C05412=1045.140,185.650,-96.102,170.888,38.031,157.175
C05413=1045.134,185.400,-96.077,170.885,38.029,157.175
C05414=1045.128,185.152,-96.053,170.883,38.027,157.174
C05415=1045.123,184.903,-96.029,170.881,38.025,157.174
C05416=1045.116,184.654,-96.006,170.877,38.023,157.173
C05417=1045.110,184.406,-95.982,170.875,38.021,157.173
C05418=1045.105,184.156,-95.958,170.873,38.019,157.173
C05419=1045.098,183.908,-95.934,170.870,38.018,157.172
C05420=1045.093,183.659,-95.909,170.868,38.017,157.172
C05421=1045.087,183.410,-95.886,170.865,38.015,157.172
C05422=1045.079,183.161,-95.863,170.863,38.013,157.171
C05423=1045.073,182.913,-95.839,170.860,38.011,157.171
C05424=1045.067,182.664,-95.815,170.858,38.010,157.171
C05425=1045.061,182.415,-95.792,170.856,38.008,157.170
C05426=1045.054,182.166,-95.768,170.852,38.007,157.170
C05427=1045.048,181.918,-95.745,170.850,38.005,157.169
C05428=1045.042,181.668,-95.721,170.848,38.004,157.169
C05429=1045.036,181.420,-95.698,170.846,38.002,157.169
C05430=1045.029,181.171,-95.674,170.843,38.000,157.168
C05431=1045.024,180.922,-95.651,170.840,37.999,157.168
C05432=1045.018,180.674,-95.627,170.838,37.997,157.168
C05433=1045.011,180.424,-95.604,170.835,37.996,157.167
C05434=1045.005,180.176,-95.580,170.833,37.994,157.167
C05435=1044.999,179.927,-95.556,170.831,37.993,157.167
C05436=1044.993,179.678,-95.533,170.828,37.991,157.166
C05437=1044.986,179.429,-95.510,170.825,37.989,157.166
C05438=1044.980,179.180,-95.487,170.823,37.988,157.165
C05439=1044.974,178.932,-95.463,170.821,37.986,157.165
C05440=1044.967,178.682,-95.440,170.818,37.984,157.165
C05441=1044.961,178.434,-95.416,170.815,37.983,157.164
C05442=1044.955,178.185,-95.393,170.813,37.982,157.164
C05443=1044.949,177.936,-95.369,170.811,37.980,157.164
C05444=1044.943,177.687,-95.346,170.808,37.979,157.163
C05445=1044.937,177.438,-95.322,170.806,37.977,157.163
C05446=1044.931,177.190,-95.299,170.804,37.975,157.163
C05447=1044.925,176.941,-95.276,170.802,37.974,157.162
C05448=1044.918,176.692,-95.253,170.798,37.972,157.162
C05449=1044.912,176.444,-95.229,170.796,37.970,157.161
C05450=1044.905,176.194,-95.206,170.794,37.969,157.161
C05451=1044.899,175.946,-95.182,170.791,37.967,157.161
C05452=1044.894,175.697,-95.159,170.789,37.966,157.160
C05453=1044.887,175.447,-95.136,170.787,37.965,157.160
C05454=1044.881,175.199,-95.112,170.784,37.963,157.160
C05455=1044.876,174.950,-95.089,170.781,37.961,157.159
C05456=1044.869,174.702,-95.066,170.779,37.960,157.159
C05457=1044.862,174.453,-95.043,170.777,37.958,157.159
C05458=1044.857,174.204,-95.020,170.774,37.956,157.158
C05459=1044.850,173.919,-94.993,170.772,37.955,157.158
C05460=1044.843,173.634,-94.967,170.769,37.953,157.158
C05461=1044.836,173.349,-94.940,170.766,37.951,157.157
C05462=1044.829,173.064,-94.913,170.763,37.949,157.157
C05463=1044.823,172.815,-94.891,170.761,37.947,157.156
C05464=1044.817,172.567,-94.868,170.759,37.946,157.156
C05465=1044.810,172.318,-94.844,170.756,37.945,157.156
C05466=1044.804,172.069,-94.821,170.754,37.943,157.155
C05467=1044.799,171.820,-94.798,170.752,37.942,157.155
C05468=1044.793,171.572,-94.774,170.749,37.940,157.155
C05469=1044.787,171.323,-94.751,170.747,37.938,157.154
C05470=1044.780,171.073,-94.728,170.744,37.937,157.154
C05471=1044.774,170.824,-94.705,170.742,37.935,157.154
C05472=1044.768,170.576,-94.682,170.739,37.933,157.153
C05473=1044.762,170.327,-94.659,170.737,37.932,157.153
C05474=1044.757,170.078,-94.636,170.735,37.930,157.153
C05475=1044.750,169.829,-94.613,170.733,37.929,157.152
C05476=1044.744,169.580,-94.590,170.730,37.927,157.152
C05477=1044.738,169.331,-94.567,170.728,37.926,157.151
C05478=1044.732,169.083,-94.544,170.726,37.925,157.151
C05479=1044.726,168.834,-94.521,170.723,37.923,157.151
C05480=1044.720,168.585,-94.497,170.721,37.921,157.150
C05481=1044.714,168.336,-94.474,170.719,37.920,157.150
C05482=1044.708,168.087,-94.452,170.717,37.918,157.150
C05483=1044.702,167.838,-94.429,170.714,37.916,157.149
C05484=1044.696,167.589,-94.406,170.712,37.915,157.149
C05485=1044.690,167.341,-94.383,170.709,37.913,157.149
C05486=1044.685,167.092,-94.360,170.707,37.912,157.148
C05487=1044.679,166.843,-94.337,170.704,37.910,157.148
C05488=1044.672,166.594,-94.314,170.702,37.909,157.148
C05489=1044.666,166.345,-94.291,170.700,37.907,157.147
C05490=1044.660,166.096,-94.268,170.697,37.906,157.147
C05491=1044.655,165.847,-94.245,170.695,37.904,157.147
C05492=1044.649,165.598,-94.222,170.693,37.903,157.146
C05493=1044.642,165.350,-94.200,170.691,37.901,157.146
C05494=1044.637,165.101,-94.177,170.688,37.900,157.146
C05495=1044.631,164.852,-94.154,170.686,37.898,157.145
C05496=1044.625,164.603,-94.131,170.684,37.896,157.145
C05497=1044.619,164.354,-94.108,170.682,37.895,157.145
C05498=1044.613,164.106,-94.086,170.679,37.893,157.144
C05499=1044.607,163.857,-94.063,170.677,37.891,157.144
C05500=1044.601,163.607,-94.039,170.675,37.890,157.144
C05501=1044.595,163.358,-94.016,170.672,37.889,157.143
C05502=1044.589,163.109,-93.993,170.670,37.887,157.143
C05503=1044.583,162.861,-93.971,170.668,37.886,157.143
C05504=1044.577,162.612,-93.948,170.666,37.884,157.142
C05505=1044.572,162.363,-93.925,170.663,37.883,157.142
C05506=1044.566,162.114,-93.902,170.661,37.881,157.142
C05507=1044.560,161.865,-93.881,170.659,37.879,157.141
C05508=1044.554,161.616,-93.858,170.657,37.878,157.141
C05509=1044.548,161.367,-93.835,170.654,37.876,157.140
C05510=1044.542,161.118,-93.812,170.652,37.875,157.140
C05511=1044.537,160.869,-93.789,170.650,37.873,157.140
C05512=1044.530,160.621,-93.767,170.647,37.871,157.139
C05513=1044.525,160.372,-93.744,170.645,37.870,157.139
C05514=1044.519,160.122,-93.721,170.643,37.868,157.139
C05515=1044.513,159.874,-93.699,170.641,37.867,157.138
C05516=1044.506,159.625,-93.677,170.638,37.865,157.138
C05517=1044.501,159.376,-93.654,170.636,37.864,157.138
C05518=1044.494,159.127,-93.632,170.634,37.863,157.138
C05519=1044.489,158.878,-93.609,170.632,37.861,157.137
C05520=1044.482,158.629,-93.587,170.629,37.860,157.137
C05521=1044.476,158.380,-93.565,170.627,37.858,157.137
C05522=1044.470,158.131,-93.542,170.625,37.857,157.136
C05523=1044.463,157.846,-93.517,170.623,37.855,157.136
C05524=1044.456,157.561,-93.491,170.620,37.854,157.136
C05525=1044.449,157.275,-93.466,170.617,37.852,157.135
C05526=1044.441,156.990,-93.440,170.615,37.851,157.135
C05527=1044.436,156.741,-93.418,170.613,37.850,157.135
C05528=1044.430,156.492,-93.395,170.610,37.848,157.134
C05529=1044.423,156.243,-93.374,170.608,37.847,157.134
C05530=1044.418,155.994,-93.351,170.606,37.845,157.134
C05531=1044.411,155.745,-93.328,170.604,37.844,157.133
C05532=1044.405,155.496,-93.307,170.601,37.842,157.133
C05533=1044.400,155.248,-93.284,170.599,37.841,157.133
C05534=1044.394,154.999,-93.262,170.597,37.839,157.132
C05535=1044.388,154.750,-93.239,170.595,37.838,157.132
C05536=1044.382,154.501,-93.218,170.592,37.837,157.132
C05537=1044.375,154.252,-93.196,170.590,37.835,157.131
C05538=1044.369,154.003,-93.174,170.588,37.834,157.131
C05539=1044.363,153.754,-93.151,170.586,37.832,157.131
C05540=1044.357,153.505,-93.129,170.583,37.831,157.131
C05541=1044.351,153.256,-93.107,170.581,37.829,157.130
C05542=1044.345,153.007,-93.085,170.579,37.828,157.130
C05543=1044.338,152.758,-93.063,170.577,37.827,157.130
C05544=1044.333,152.509,-93.041,170.574,37.825,157.129
C05545=1044.326,152.260,-93.018,170.572,37.824,157.129
C05546=1044.320,152.011,-92.997,170.570,37.823,157.129
C05547=1044.314,151.762,-92.974,170.569,37.821,157.128
C05548=1044.308,151.513,-92.952,170.567,37.820,157.128
C05549=1044.302,151.264,-92.931,170.564,37.819,157.128
C05550=1044.296,151.016,-92.909,170.562,37.817,157.127
C05551=1044.290,150.767,-92.887,170.560,37.816,157.127
C05552=1044.284,150.518,-92.865,170.558,37.815,157.127
C05553=1044.278,150.269,-92.842,170.555,37.813,157.126
C05554=1044.272,150.019,-92.821,170.553,37.812,157.126
C05555=1044.266,149.771,-92.798,170.551,37.810,157.126
C05556=1044.259,149.522,-92.777,170.549,37.809,157.126
C05557=1044.253,149.272,-92.755,170.546,37.808,157.125
C05558=1044.247,149.024,-92.733,170.544,37.806,157.125
C05559=1044.242,148.775,-92.711,170.542,37.805,157.125
C05560=1044.236,148.526,-92.689,170.540,37.803,157.124
C05561=1044.230,148.277,-92.668,170.538,37.802,157.124
C05562=1044.223,148.028,-92.645,170.535,37.801,157.124
C05563=1044.217,147.779,-92.624,170.533,37.799,157.123
C05564=1044.211,147.530,-92.602,170.532,37.798,157.123
C05565=1044.205,147.280,-92.580,170.530,37.797,157.123
C05566=1044.199,147.032,-92.558,170.527,37.796,157.123
C05567=1044.193,146.783,-92.537,170.525,37.794,157.122
C05568=1044.186,146.534,-92.515,170.523,37.793,157.122
C05569=1044.180,146.285,-92.493,170.521,37.792,157.122
C05570=1044.174,146.036,-92.472,170.518,37.790,157.122
C05571=1044.168,145.787,-92.449,170.516,37.789,157.121
C05572=1044.161,145.538,-92.428,170.514,37.787,157.121
C05573=1044.156,145.289,-92.407,170.512,37.786,157.121
C05574=1044.150,145.040,-92.385,170.510,37.785,157.120
C05575=1044.144,144.791,-92.363,170.507,37.784,157.120
C05576=1044.137,144.542,-92.342,170.505,37.783,157.120
C05577=1044.131,144.293,-92.320,170.503,37.781,157.119
C05578=1044.125,144.045,-92.298,170.502,37.780,157.119
C05579=1044.119,143.795,-92.276,170.499,37.778,157.119
C05580=1044.113,143.546,-92.255,170.497,37.777,157.119
C05581=1044.107,143.297,-92.233,170.495,37.775,157.118
C05582=1044.101,143.048,-92.211,170.493,37.774,157.118
C05583=1044.095,142.799,-92.190,170.491,37.773,157.118
C05584=1044.089,142.550,-92.169,170.488,37.772,157.117
C05585=1044.082,142.301,-92.148,170.486,37.771,157.117
C05586=1044.076,142.052,-92.126,170.484,37.769,157.117
C05587=1044.069,141.767,-92.101,170.482,37.768,157.117
C05588=1044.063,141.481,-92.076,170.479,37.766,157.116
C05589=1044.056,141.195,-92.051,170.477,37.765,157.116
C05590=1044.048,140.909,-92.027,170.475,37.763,157.116
C05591=1044.043,140.661,-92.006,170.473,37.762,157.115
C05592=1044.037,140.412,-91.984,170.470,37.761,157.115
C05593=1044.030,140.162,-91.963,170.468,37.759,157.115
C05594=1044.024,139.913,-91.941,170.466,37.758,157.114
C05595=1044.019,139.665,-91.920,170.464,37.757,157.114
C05596=1044.013,139.416,-91.898,170.462,37.755,157.114
C05597=1044.006,139.166,-91.877,170.459,37.754,157.114
C05598=1043.999,138.917,-91.856,170.458,37.753,157.113
C05599=1043.994,138.669,-91.834,170.456,37.751,157.113
C05600=1043.988,138.420,-91.813,170.454,37.750,157.113
C05601=1043.982,138.170,-91.791,170.451,37.749,157.112
C05602=1043.975,137.922,-91.770,170.449,37.748,157.112
C05603=1043.969,137.672,-91.749,170.447,37.746,157.112
C05604=1043.963,137.423,-91.728,170.445,37.745,157.112
C05605=1043.957,137.174,-91.706,170.443,37.744,157.111
C05606=1043.951,136.926,-91.685,170.441,37.742,157.111
C05607=1043.945,136.677,-91.664,170.439,37.741,157.111
C05608=1043.939,136.427,-91.643,170.437,37.740,157.110
C05609=1043.933,136.179,-91.622,170.435,37.739,157.110
C05610=1043.926,135.929,-91.601,170.433,37.737,157.110
C05611=1043.920,135.680,-91.579,170.430,37.736,157.110
C05612=1043.914,135.431,-91.557,170.428,37.735,157.109
C05613=1043.908,135.182,-91.537,170.426,37.734,157.109
C05614=1043.902,134.933,-91.516,170.425,37.733,157.109
C05615=1043.896,134.684,-91.494,170.422,37.731,157.109
C05616=1043.889,134.436,-91.473,170.420,37.730,157.108
C05617=1043.884,134.186,-91.453,170.418,37.729,157.108
C05618=1043.878,133.937,-91.431,170.416,37.727,157.108
C05619=1043.871,133.688,-91.410,170.414,37.726,157.107
C05620=1043.865,133.439,-91.389,170.411,37.725,157.107
C05621=1043.860,133.190,-91.368,170.410,37.724,157.107
C05622=1043.853,132.941,-91.347,170.408,37.723,157.107
C05623=1043.847,132.692,-91.325,170.406,37.721,157.106
C05624=1043.841,132.443,-91.305,170.404,37.720,157.106
C05625=1043.834,132.194,-91.284,170.401,37.718,157.106
C05626=1043.828,131.945,-91.262,170.399,37.717,157.106
C05627=1043.823,131.696,-91.242,170.397,37.716,157.105
C05628=1043.816,131.447,-91.221,170.396,37.715,157.105
C05629=1043.811,131.198,-91.200,170.394,37.714,157.105
C05630=1043.804,130.949,-91.179,170.391,37.712,157.104
C05631=1043.798,130.699,-91.157,170.389,37.711,157.104
C05632=1043.792,130.451,-91.137,170.387,37.710,157.104
C05633=1043.785,130.202,-91.116,170.385,37.709,157.104
C05634=1043.779,129.952,-91.095,170.383,37.708,157.103
C05635=1043.773,129.704,-91.075,170.381,37.707,157.103
C05636=1043.767,129.454,-91.054,170.379,37.705,157.103
C05637=1043.760,129.205,-91.033,170.377,37.704,157.103
C05638=1043.754,128.956,-91.013,170.375,37.703,157.102
C05639=1043.748,128.707,-90.991,170.373,37.702,157.102
C05640=1043.742,128.458,-90.971,170.370,37.701,157.102
C05641=1043.735,128.209,-90.950,170.368,37.699,157.102
C05642=1043.729,127.959,-90.929,170.367,37.698,157.101
C05643=1043.723,127.711,-90.909,170.365,37.697,157.101
C05644=1043.716,127.462,-90.888,170.363,37.696,157.101
C05645=1043.711,127.213,-90.868,170.360,37.695,157.101
C05646=1043.704,126.964,-90.847,170.358,37.693,157.100
C05647=1043.698,126.714,-90.826,170.356,37.692,157.100
C05648=1043.692,126.466,-90.805,170.354,37.691,157.100
C05649=1043.685,126.216,-90.785,170.353,37.690,157.100
C05650=1043.680,125.967,-90.764,170.350,37.689,157.099
C05651=1043.672,125.681,-90.740,170.348,37.687,157.099
C05652=1043.665,125.396,-90.716,170.346,37.686,157.099
C05653=1043.658,125.110,-90.692,170.343,37.685,157.098
C05654=1043.651,124.824,-90.669,170.341,37.683,157.098
C05655=1043.645,124.575,-90.649,170.339,37.682,157.098
C05656=1043.639,124.325,-90.628,170.337,37.681,157.098
C05657=1043.633,124.077,-90.607,170.335,37.680,157.097
C05658=1043.626,123.828,-90.587,170.333,37.679,157.097
C05659=1043.620,123.578,-90.566,170.331,37.677,157.097
C05660=1043.614,123.330,-90.545,170.328,37.676,157.097
C05661=1043.607,123.080,-90.525,170.327,37.675,157.096
C05662=1043.602,122.831,-90.504,170.325,37.674,157.096
C05663=1043.595,122.582,-90.484,170.323,37.673,157.096
C05664=1043.589,122.333,-90.463,170.321,37.671,157.096
C05665=1043.583,122.085,-90.443,170.318,37.670,157.095
C05666=1043.577,121.835,-90.423,170.317,37.669,157.095
C05667=1043.571,121.587,-90.402,170.315,37.668,157.095
C05668=1043.564,121.337,-90.382,170.313,37.667,157.095
C05669=1043.559,121.088,-90.361,170.311,37.665,157.094
C05670=1043.553,120.838,-90.341,170.308,37.664,157.094
C05671=1043.547,120.590,-90.321,170.307,37.663,157.094
C05672=1043.540,120.340,-90.299,170.305,37.662,157.093
C05673=1043.534,120.092,-90.279,170.303,37.661,157.093
C05674=1043.528,119.842,-90.259,170.301,37.659,157.093
C05675=1043.523,119.593,-90.238,170.298,37.658,157.093
C05676=1043.516,119.345,-90.218,170.297,37.657,157.092
C05677=1043.510,119.095,-90.197,170.295,37.656,157.092
C05678=1043.504,118.846,-90.177,170.293,37.655,157.092
C05679=1043.498,118.597,-90.156,170.291,37.653,157.092
C05680=1043.492,118.348,-90.136,170.288,37.652,157.091
C05681=1043.485,118.098,-90.116,170.287,37.651,157.091
C05682=1043.480,117.849,-90.096,170.285,37.650,157.091
C05683=1043.474,117.601,-90.075,170.283,37.649,157.091
C05684=1043.467,117.351,-90.055,170.281,37.647,157.090
C05685=1043.461,117.103,-90.035,170.280,37.646,157.090
C05686=1043.456,116.854,-90.014,170.277,37.645,157.090
C05687=1043.449,116.604,-89.994,170.275,37.644,157.090
C05688=1043.443,116.355,-89.974,170.273,37.643,157.089
C05689=1043.437,116.105,-89.953,170.271,37.641,157.089
C05690=1043.431,115.857,-89.933,170.269,37.640,157.089
C05691=1043.425,115.608,-89.913,170.267,37.638,157.088
C05692=1043.419,115.358,-89.893,170.265,37.637,157.088
C05693=1043.413,115.110,-89.871,170.263,37.636,157.088
C05694=1043.407,114.861,-89.851,170.262,37.635,157.088
C05695=1043.401,114.611,-89.831,170.259,37.634,157.087
C05696=1043.395,114.363,-89.811,170.257,37.632,157.087
C05697=1043.389,114.113,-89.791,170.255,37.631,157.087
C05698=1043.383,113.864,-89.770,170.254,37.630,157.087
C05699=1043.377,113.615,-89.750,170.252,37.629,157.086
C05700=1043.371,113.366,-89.730,170.250,37.628,157.086
C05701=1043.364,113.117,-89.710,170.247,37.626,157.086
C05702=1043.358,112.868,-89.690,170.246,37.625,157.086
C05703=1043.353,112.619,-89.671,170.244,37.624,157.085
C05704=1043.346,112.369,-89.650,170.242,37.623,157.085
C05705=1043.340,112.120,-89.630,170.240,37.622,157.085
C05706=1043.333,111.871,-89.610,170.237,37.621,157.085
C05707=1043.327,111.622,-89.590,170.236,37.620,157.085
C05708=1043.321,111.373,-89.570,170.234,37.619,157.084
C05709=1043.315,111.124,-89.550,170.232,37.617,157.084
C05710=1043.309,110.875,-89.530,170.230,37.616,157.084
C05711=1043.303,110.626,-89.510,170.228,37.615,157.083
C05712=1043.296,110.376,-89.490,170.226,37.614,157.083
C05713=1043.290,110.127,-89.470,170.224,37.613,157.083
C05714=1043.284,109.878,-89.450,170.222,37.611,157.083
C05715=1043.278,109.592,-89.428,170.220,37.610,157.082
C05716=1043.270,109.306,-89.405,170.218,37.609,157.082
C05717=1043.263,109.020,-89.382,170.215,37.608,157.082
C05718=1043.256,108.734,-89.360,170.213,37.607,157.082
C05719=1043.250,108.485,-89.340,170.211,37.605,157.081
C05720=1043.243,108.236,-89.319,170.209,37.604,157.081
C05721=1043.237,107.986,-89.300,170.208,37.603,157.081
C05722=1043.231,107.737,-89.280,170.205,37.602,157.081
C05723=1043.224,107.488,-89.260,170.203,37.601,157.081
C05724=1043.218,107.239,-89.240,170.201,37.600,157.080
C05725=1043.212,106.990,-89.221,170.200,37.599,157.080
C05726=1043.206,106.741,-89.201,170.198,37.598,157.080
C05727=1043.200,106.492,-89.181,170.195,37.596,157.079
C05728=1043.194,106.243,-89.161,170.193,37.595,157.079
C05729=1043.188,105.993,-89.142,170.192,37.594,157.079
C05730=1043.181,105.745,-89.122,170.190,37.593,157.079
C05731=1043.175,105.495,-89.102,170.188,37.592,157.079
C05732=1043.169,105.246,-89.083,170.186,37.591,157.078
C05733=1043.163,104.997,-89.063,170.183,37.590,157.078
C05734=1043.157,104.748,-89.043,170.182,37.589,157.078
C05735=1043.151,104.498,-89.023,170.180,37.587,157.078
C05736=1043.144,104.250,-89.004,170.178,37.586,157.077
C05737=1043.138,104.000,-88.985,170.176,37.585,157.077
C05738=1043.132,103.751,-88.965,170.174,37.584,157.077
C05739=1043.126,103.502,-88.944,170.172,37.583,157.077
C05740=1043.120,103.253,-88.925,170.170,37.582,157.076
C05741=1043.113,103.004,-88.906,170.168,37.581,157.076
C05742=1043.108,102.755,-88.886,170.167,37.580,157.076
C05743=1043.102,102.506,-88.866,170.165,37.578,157.076
C05744=1043.095,102.256,-88.846,170.162,37.577,157.075
C05745=1043.089,102.007,-88.827,170.160,37.576,157.075
C05746=1043.083,101.758,-88.808,170.159,37.575,157.075
C05747=1043.077,101.509,-88.788,170.157,37.574,157.075
C05748=1043.071,101.260,-88.768,170.155,37.572,157.074
C05749=1043.065,101.010,-88.749,170.154,37.572,157.074
C05750=1043.059,100.761,-88.729,170.151,37.571,157.074
C05751=1043.052,100.512,-88.710,170.149,37.569,157.074
C05752=1043.046,100.263,-88.690,170.147,37.568,157.073
C05753=1043.041,100.014,-88.671,170.146,37.567,157.073
C05754=1043.033,99.765,-88.651,170.144,37.566,157.073
C05755=1043.028,99.515,-88.632,170.142,37.565,157.073
C05756=1043.021,99.267,-88.613,170.139,37.564,157.073
C05757=1043.015,99.017,-88.593,170.137,37.563,157.072
C05758=1043.008,98.769,-88.574,170.136,37.562,157.072
C05759=1043.002,98.519,-88.554,170.134,37.561,157.072
C05760=1042.996,98.269,-88.535,170.132,37.560,157.072
C05761=1042.990,98.021,-88.516,170.129,37.559,157.071
C05762=1042.984,97.771,-88.496,170.128,37.557,157.071
C05763=1042.977,97.523,-88.477,170.126,37.556,157.071
C05764=1042.972,97.273,-88.458,170.124,37.556,157.071
C05765=1042.965,97.023,-88.439,170.122,37.554,157.071
C05766=1042.959,96.775,-88.419,170.121,37.553,157.070
C05767=1042.952,96.525,-88.400,170.118,37.552,157.070
C05768=1042.946,96.276,-88.381,170.116,37.551,157.070
C05769=1042.940,96.028,-88.362,170.114,37.550,157.070
C05770=1042.934,95.778,-88.342,170.113,37.549,157.069
C05771=1042.928,95.529,-88.323,170.111,37.548,157.069
C05772=1042.921,95.279,-88.303,170.109,37.547,157.069
C05773=1042.915,95.030,-88.284,170.106,37.545,157.069
C05774=1042.909,94.781,-88.266,170.105,37.545,157.069
C05775=1042.903,94.532,-88.246,170.103,37.544,157.068
C05776=1042.896,94.283,-88.227,170.101,37.542,157.068
C05777=1042.891,94.034,-88.208,170.099,37.541,157.068
C05778=1042.884,93.784,-88.189,170.098,37.540,157.067
C05779=1042.877,93.499,-88.167,170.095,37.539,157.067
C05780=1042.871,93.212,-88.144,170.093,37.537,157.067
C05781=1042.863,92.926,-88.122,170.091,37.536,157.067
C05782=1042.856,92.640,-88.101,170.089,37.535,157.066
C05783=1042.850,92.391,-88.082,170.087,37.534,157.066
C05784=1042.844,92.142,-88.062,170.084,37.533,157.066
C05785=1042.837,91.893,-88.043,170.083,37.532,157.066
C05786=1042.831,91.644,-88.024,170.081,37.531,157.066
C05787=1042.825,91.394,-88.005,170.079,37.530,157.065
C05788=1042.819,91.145,-87.986,170.077,37.528,157.065
C05789=1042.813,90.897,-87.967,170.076,37.527,157.065
C05790=1042.807,90.647,-87.948,170.073,37.526,157.065
C05791=1042.800,90.398,-87.929,170.071,37.525,157.064
C05792=1042.795,90.149,-87.910,170.070,37.524,157.064
C05793=1042.788,89.899,-87.891,170.068,37.523,157.064
C05794=1042.782,89.650,-87.872,170.066,37.522,157.064
C05795=1042.776,89.400,-87.853,170.064,37.521,157.064
C05796=1042.769,89.151,-87.834,170.061,37.520,157.063
C05797=1042.763,88.902,-87.815,170.060,37.519,157.063
C05798=1042.756,88.653,-87.797,170.058,37.518,157.063
C05799=1042.750,88.404,-87.777,170.056,37.517,157.063
C05800=1042.744,88.155,-87.758,170.054,37.516,157.062
C05801=1042.737,87.906,-87.740,170.053,37.515,157.062
C05802=1042.731,87.657,-87.721,170.050,37.514,157.062
C05803=1042.725,87.407,-87.702,170.048,37.513,157.062
C05804=1042.719,87.158,-87.683,170.046,37.512,157.061
C05805=1042.713,86.909,-87.664,170.045,37.511,157.061
C05806=1042.706,86.660,-87.646,170.043,37.510,157.061
C05807=1042.700,86.410,-87.626,170.041,37.509,157.061
C05808=1042.694,86.161,-87.608,170.039,37.507,157.061
C05809=1042.688,85.912,-87.589,170.037,37.507,157.060
C05810=1042.681,85.663,-87.570,170.035,37.506,157.060
C05811=1042.675,85.414,-87.552,170.033,37.504,157.060
C05812=1042.669,85.164,-87.533,170.032,37.504,157.060
C05813=1042.663,84.915,-87.515,170.030,37.503,157.060
C05814=1042.656,84.666,-87.496,170.028,37.501,157.059
C05815=1042.650,84.416,-87.477,170.025,37.500,157.059
C05816=1042.644,84.167,-87.458,170.024,37.499,157.059
C05817=1042.638,83.918,-87.439,170.022,37.498,157.059
C05818=1042.632,83.669,-87.421,170.020,37.497,157.058
C05819=1042.625,83.420,-87.402,170.018,37.496,157.058
C05820=1042.619,83.171,-87.384,170.017,37.495,157.058
C05821=1042.613,82.921,-87.364,170.014,37.494,157.058
C05822=1042.607,82.672,-87.346,170.012,37.493,157.058
C05823=1042.600,82.423,-87.327,170.010,37.492,157.057
C05824=1042.594,82.173,-87.309,170.009,37.491,157.057
C05825=1042.588,81.924,-87.290,170.007,37.490,157.057
C05826=1042.582,81.675,-87.271,170.005,37.489,157.057
C05827=1042.575,81.425,-87.253,170.003,37.487,157.056
C05828=1042.570,81.177,-87.234,170.001,37.487,157.056
C05829=1042.563,80.928,-87.216,169.999,37.486,157.056
C05830=1042.557,80.678,-87.198,169.997,37.484,157.056
C05831=1042.551,80.429,-87.178,169.996,37.483,157.056
C05832=1042.545,80.180,-87.160,169.994,37.483,157.055
C05833=1042.539,79.931,-87.141,169.991,37.481,157.055
C05834=1042.532,79.681,-87.122,169.990,37.480,157.055
C05835=1042.526,79.432,-87.105,169.988,37.479,157.055
C05836=1042.520,79.182,-87.085,169.986,37.478,157.055
C05837=1042.514,78.933,-87.067,169.984,37.477,157.054
C05838=1042.508,78.685,-87.048,169.983,37.476,157.054
C05839=1042.502,78.436,-87.030,169.980,37.475,157.054
C05840=1042.496,78.186,-87.012,169.978,37.474,157.054
C05841=1042.489,77.937,-86.993,169.976,37.473,157.053
C05842=1042.483,77.688,-86.974,169.975,37.472,157.053
C05843=1042.476,77.401,-86.954,169.973,37.470,157.053
C05844=1042.469,77.115,-86.933,169.971,37.469,157.053
C05845=1042.461,76.829,-86.911,169.968,37.468,157.052
C05846=1042.454,76.543,-86.890,169.966,37.467,157.052
C05847=1042.448,76.295,-86.872,169.964,37.466,157.052
C05848=1042.442,76.045,-86.854,169.962,37.465,157.052
C05849=1042.435,75.796,-86.835,169.961,37.464,157.051
C05850=1042.429,75.546,-86.817,169.959,37.463,157.051
C05851=1042.423,75.297,-86.799,169.956,37.462,157.051
C05852=1042.416,75.048,-86.780,169.954,37.461,157.051
C05853=1042.410,74.798,-86.762,169.953,37.460,157.051
C05854=1042.404,74.549,-86.744,169.951,37.459,157.050
C05855=1042.398,74.300,-86.726,169.949,37.458,157.050
C05856=1042.392,74.051,-86.707,169.947,37.457,157.050
C05857=1042.385,73.802,-86.689,169.946,37.456,157.050
C05858=1042.379,73.552,-86.671,169.943,37.455,157.050
C05859=1042.372,73.303,-86.653,169.941,37.454,157.049
C05860=1042.366,73.053,-86.635,169.939,37.453,157.049
C05861=1042.360,72.805,-86.616,169.938,37.452,157.049
C05862=1042.354,72.555,-86.599,169.936,37.451,157.049
C05863=1042.348,72.306,-86.580,169.934,37.450,157.049
C05864=1042.341,72.056,-86.562,169.931,37.449,157.048
C05865=1042.335,71.807,-86.543,169.930,37.448,157.048
C05866=1042.329,71.558,-86.526,169.928,37.447,157.048
C05867=1042.323,71.309,-86.507,169.926,37.446,157.048
C05868=1042.317,71.059,-86.489,169.925,37.445,157.048
C05869=1042.310,70.810,-86.471,169.923,37.444,157.047
C05870=1042.304,70.561,-86.453,169.920,37.443,157.047
C05871=1042.298,70.312,-86.435,169.918,37.442,157.047
C05872=1042.292,70.062,-86.417,169.917,37.441,157.047
C05873=1042.285,69.813,-86.398,169.915,37.440,157.046
C05874=1042.279,69.564,-86.380,169.913,37.439,157.046
C05875=1042.273,69.314,-86.362,169.911,37.438,157.046
C05876=1042.266,69.066,-86.345,169.910,37.437,157.046
C05877=1042.260,68.816,-86.327,169.907,37.436,157.046
C05878=1042.254,68.567,-86.308,169.905,37.435,157.045
C05879=1042.248,68.317,-86.290,169.903,37.434,157.045
C05880=1042.242,68.068,-86.273,169.902,37.433,157.045
C05881=1042.235,67.819,-86.255,169.900,37.432,157.045
C05882=1042.229,67.570,-86.237,169.898,37.431,157.045
C05883=1042.223,67.320,-86.219,169.896,37.430,157.044
C05884=1042.216,67.071,-86.201,169.894,37.429,157.044
C05885=1042.210,66.822,-86.183,169.892,37.428,157.044
C05886=1042.204,66.572,-86.165,169.890,37.427,157.044
C05887=1042.198,66.323,-86.147,169.888,37.426,157.044
C05888=1042.191,66.074,-86.129,169.887,37.425,157.043
C05889=1042.185,65.825,-86.112,169.885,37.424,157.043
C05890=1042.179,65.576,-86.093,169.883,37.423,157.043
C05891=1042.172,65.326,-86.076,169.880,37.422,157.043
C05892=1042.166,65.077,-86.058,169.879,37.421,157.043
C05893=1042.160,64.827,-86.040,169.877,37.420,157.042
C05894=1042.153,64.579,-86.022,169.875,37.419,157.042
C05895=1042.147,64.329,-86.004,169.873,37.418,157.042
C05896=1042.142,64.080,-85.987,169.872,37.417,157.042
C05897=1042.135,63.830,-85.969,169.869,37.416,157.041
C05898=1042.129,63.581,-85.951,169.867,37.415,157.041
C05899=1042.121,63.332,-85.933,169.865,37.415,157.041
C05900=1042.116,63.083,-85.916,169.864,37.413,157.041
C05901=1042.109,62.833,-85.898,169.862,37.413,157.041
C05902=1042.102,62.584,-85.881,169.860,37.412,157.041
C05903=1042.096,62.334,-85.863,169.858,37.411,157.040
C05904=1042.090,62.085,-85.846,169.857,37.410,157.040
C05905=1042.083,61.836,-85.827,169.854,37.409,157.040
C05906=1042.076,61.587,-85.810,169.852,37.408,157.040
C05907=1042.070,61.301,-85.790,169.850,37.407,157.040
C05908=1042.062,61.014,-85.770,169.848,37.406,157.039
C05909=1042.055,60.728,-85.750,169.846,37.405,157.039
C05910=1042.047,60.442,-85.730,169.844,37.404,157.039
C05911=1042.041,60.192,-85.712,169.842,37.403,157.039
C05912=1042.035,59.943,-85.695,169.839,37.402,157.039
C05913=1042.028,59.694,-85.677,169.838,37.401,157.038
C05914=1042.022,59.444,-85.659,169.836,37.400,157.038
C05915=1042.016,59.195,-85.642,169.834,37.400,157.038
C05916=1042.009,58.946,-85.625,169.832,37.398,157.038
C05917=1042.003,58.696,-85.607,169.830,37.398,157.038
C05918=1041.996,58.447,-85.590,169.829,37.397,157.037
C05919=1041.990,58.198,-85.573,169.826,37.396,157.037
C05920=1041.984,57.948,-85.555,169.824,37.395,157.037
C05921=1041.977,57.700,-85.538,169.822,37.394,157.037
C05922=1041.971,57.450,-85.520,169.821,37.393,157.037
C05923=1041.964,57.200,-85.503,169.819,37.392,157.037
C05924=1041.958,56.952,-85.486,169.817,37.391,157.036
C05925=1041.952,56.702,-85.468,169.815,37.391,157.036
C05926=1041.945,56.452,-85.450,169.813,37.389,157.036
C05927=1041.940,56.203,-85.433,169.811,37.389,157.036
C05928=1041.933,55.954,-85.416,169.809,37.387,157.036
C05929=1041.926,55.705,-85.398,169.807,37.387,157.035
C05930=1041.920,55.455,-85.381,169.805,37.386,157.035
C05931=1041.914,55.206,-85.363,169.804,37.385,157.035
C05932=1041.907,54.957,-85.346,169.802,37.384,157.035
C05933=1041.901,54.708,-85.328,169.799,37.383,157.035
C05934=1041.894,54.458,-85.311,169.797,37.382,157.034
C05935=1041.889,54.209,-85.294,169.796,37.381,157.034
C05936=1041.882,53.959,-85.277,169.794,37.380,157.034
C05937=1041.876,53.710,-85.260,169.792,37.379,157.034
C05938=1041.870,53.461,-85.242,169.790,37.378,157.034
C05939=1041.864,53.212,-85.225,169.789,37.377,157.033
C05940=1041.857,52.962,-85.208,169.787,37.377,157.033
C05941=1041.851,52.713,-85.190,169.784,37.375,157.033
C05942=1041.844,52.464,-85.173,169.782,37.375,157.033
C05943=1041.839,52.214,-85.156,169.780,37.373,157.033
C05944=1041.832,51.965,-85.139,169.779,37.372,157.032
C05945=1041.825,51.715,-85.121,169.777,37.372,157.032
C05946=1041.820,51.466,-85.104,169.775,37.370,157.032
C05947=1041.813,51.217,-85.086,169.773,37.370,157.032
C05948=1041.807,50.968,-85.069,169.771,37.369,157.032
C05949=1041.801,50.718,-85.052,169.769,37.368,157.032
C05950=1041.795,50.469,-85.035,169.767,37.367,157.031
C05951=1041.788,50.220,-85.018,169.765,37.366,157.031
C05952=1041.782,49.971,-85.000,169.764,37.365,157.031
C05953=1041.776,49.721,-84.984,169.762,37.364,157.031
C05954=1041.770,49.472,-84.967,169.760,37.363,157.031
C05955=1041.763,49.222,-84.949,169.757,37.362,157.030
C05956=1041.757,48.973,-84.932,169.756,37.361,157.030
C05957=1041.751,48.723,-84.915,169.754,37.360,157.030
C05958=1041.745,48.474,-84.898,169.752,37.359,157.030
C05959=1041.738,48.225,-84.880,169.750,37.358,157.029
C05960=1041.732,47.976,-84.863,169.749,37.357,157.029
C05961=1041.726,47.726,-84.846,169.747,37.356,157.029
C05962=1041.720,47.477,-84.829,169.744,37.355,157.029
C05963=1041.713,47.228,-84.812,169.742,37.355,157.029
C05964=1041.708,46.978,-84.795,169.740,37.353,157.028
C05965=1041.702,46.729,-84.778,169.739,37.352,157.028
C05966=1041.695,46.480,-84.761,169.737,37.352,157.028
C05967=1041.690,46.230,-84.744,169.735,37.350,157.028
C05968=1041.683,45.981,-84.726,169.733,37.350,157.028
C05969=1041.676,45.732,-84.709,169.731,37.348,157.027
C05970=1041.671,45.482,-84.692,169.729,37.347,157.027
C05971=1041.663,45.196,-84.673,169.727,37.347,157.027
C05972=1041.656,44.909,-84.654,169.725,37.345,157.027
C05973=1041.649,44.623,-84.633,169.723,37.344,157.027
C05974=1041.642,44.336,-84.614,169.721,37.343,157.026
C05975=1041.635,44.087,-84.597,169.718,37.342,157.026
C05976=1041.630,43.837,-84.580,169.716,37.341,157.026
C05977=1041.624,43.588,-84.563,169.715,37.340,157.026
C05978=1041.617,43.338,-84.546,169.713,37.339,157.026
C05979=1041.611,43.090,-84.529,169.711,37.338,157.025
C05980=1041.604,42.840,-84.513,169.709,37.337,157.025
C05981=1041.599,42.591,-84.495,169.707,37.336,157.025
C05982=1041.593,42.341,-84.479,169.705,37.336,157.025
C05983=1041.586,42.092,-84.462,169.703,37.334,157.025
C05984=1041.580,41.842,-84.445,169.701,37.334,157.024
C05985=1041.573,41.593,-84.428,169.699,37.333,157.024
C05986=1041.567,41.344,-84.412,169.697,37.332,157.024
C05987=1041.561,41.095,-84.395,169.696,37.331,157.024
C05988=1041.554,40.845,-84.378,169.694,37.330,157.024
C05989=1041.548,40.596,-84.361,169.692,37.329,157.023
C05990=1041.542,40.346,-84.344,169.689,37.328,157.023
C05991=1041.536,40.097,-84.328,169.687,37.328,157.023
C05992=1041.529,39.848,-84.311,169.686,37.327,157.023
C05993=1041.523,39.598,-84.295,169.684,37.326,157.023
C05994=1041.517,39.349,-84.278,169.682,37.325,157.023
C05995=1041.511,39.100,-84.261,169.680,37.324,157.022
C05996=1041.504,38.851,-84.244,169.678,37.323,157.022
C05997=1041.498,38.601,-84.228,169.677,37.322,157.022
C05998=1041.491,38.351,-84.211,169.674,37.321,157.022
C05999=1041.485,38.102,-84.194,169.672,37.320,157.022
C06000=1041.479,37.853,-84.178,169.670,37.319,157.021
C06001=1041.473,37.603,-84.161,169.668,37.319,157.021
C06002=1041.466,37.354,-84.144,169.667,37.317,157.021
C06003=1041.460,37.105,-84.128,169.665,37.317,157.021
C06004=1041.454,36.855,-84.111,169.663,37.316,157.021
C06005=1041.447,36.606,-84.094,169.660,37.315,157.021
C06006=1041.442,36.357,-84.078,169.658,37.314,157.020
C06007=1041.435,36.107,-84.062,169.657,37.313,157.020
C06008=1041.428,35.858,-84.046,169.655,37.312,157.020
C06009=1041.422,35.609,-84.029,169.653,37.312,157.020
C06010=1041.415,35.359,-84.012,169.651,37.311,157.020
C06011=1041.410,35.110,-83.996,169.649,37.310,157.020
C06012=1041.404,34.860,-83.980,169.647,37.309,157.019
C06013=1041.397,34.611,-83.963,169.645,37.308,157.019
C06014=1041.390,34.362,-83.947,169.643,37.308,157.019
C06015=1041.384,34.112,-83.931,169.641,37.306,157.019
C06016=1041.378,33.862,-83.914,169.639,37.306,157.019
C06017=1041.372,33.613,-83.898,169.637,37.305,157.018
C06018=1041.365,33.364,-83.881,169.635,37.304,157.018
C06019=1041.358,33.115,-83.865,169.634,37.303,157.018
C06020=1041.352,32.865,-83.848,169.632,37.302,157.018
C06021=1041.346,32.616,-83.832,169.629,37.302,157.018
C06022=1041.340,32.366,-83.816,169.627,37.300,157.018
C06023=1041.333,32.117,-83.799,169.625,37.300,157.017
C06024=1041.327,31.868,-83.783,169.624,37.299,157.017
C06025=1041.321,31.619,-83.767,169.622,37.298,157.017
C06026=1041.314,31.369,-83.750,169.620,37.297,157.017
C06027=1041.308,31.119,-83.734,169.618,37.296,157.017
C06028=1041.302,30.870,-83.718,169.616,37.295,157.017
C06029=1041.296,30.621,-83.702,169.614,37.295,157.016
C06030=1041.289,30.371,-83.685,169.612,37.294,157.016
C06031=1041.283,30.122,-83.668,169.610,37.293,157.016
C06032=1041.277,29.873,-83.652,169.608,37.292,157.016
C06033=1041.270,29.624,-83.636,169.606,37.291,157.016
C06034=1041.264,29.374,-83.620,169.604,37.291,157.016
C06035=1041.257,29.086,-83.601,169.602,37.289,157.015
C06036=1041.250,28.800,-83.583,169.600,37.288,157.015
C06037=1041.242,28.514,-83.564,169.597,37.288,157.015
C06038=1041.235,28.228,-83.545,169.595,37.286,157.015
C06039=1041.229,27.978,-83.529,169.593,37.286,157.015
C06040=1041.223,27.728,-83.512,169.591,37.285,157.014
C06041=1041.216,27.479,-83.497,169.589,37.284,157.014
C06042=1041.210,27.229,-83.481,169.587,37.283,157.014
C06043=1041.203,26.980,-83.466,169.586,37.283,157.014
C06044=1041.197,26.730,-83.449,169.584,37.281,157.014
C06045=1041.191,26.481,-83.433,169.581,37.281,157.014
C06046=1041.184,26.232,-83.417,169.579,37.280,157.013
C06047=1041.178,25.983,-83.401,169.577,37.279,157.013
C06048=1041.172,25.733,-83.385,169.575,37.278,157.013
C06049=1041.165,25.483,-83.368,169.573,37.278,157.013
C06050=1041.159,25.234,-83.352,169.572,37.277,157.013
C06051=1041.152,24.985,-83.337,169.570,37.276,157.013
C06052=1041.147,24.736,-83.320,169.568,37.275,157.012
C06053=1041.140,24.487,-83.305,169.565,37.274,157.012
C06054=1041.133,24.237,-83.288,169.563,37.273,157.012
C06055=1041.127,23.987,-83.273,169.561,37.273,157.012
C06056=1041.121,23.738,-83.257,169.559,37.272,157.012
C06057=1041.114,23.489,-83.241,169.557,37.271,157.012
C06058=1041.108,23.239,-83.225,169.556,37.270,157.011
C06059=1041.102,22.990,-83.209,169.554,37.269,157.011
C06060=1041.095,22.740,-83.193,169.552,37.269,157.011
C06061=1041.089,22.490,-83.177,169.550,37.268,157.011
C06062=1041.083,22.241,-83.161,169.548,37.267,157.011
C06063=1041.077,21.992,-83.145,169.545,37.266,157.011
C06064=1041.070,21.743,-83.129,169.543,37.266,157.010
C06065=1041.064,21.493,-83.113,169.542,37.265,157.010
C06066=1041.058,21.244,-83.098,169.540,37.264,157.010
C06067=1041.052,20.994,-83.082,169.538,37.263,157.010
C06068=1041.045,20.745,-83.066,169.536,37.263,157.010
C06069=1041.039,20.495,-83.050,169.534,37.261,157.010
C06070=1041.032,20.246,-83.034,169.532,37.261,157.009
C06071=1041.026,19.996,-83.019,169.529,37.260,157.009
C06072=1041.020,19.747,-83.003,169.527,37.259,157.009
C06073=1041.014,19.498,-82.987,169.526,37.258,157.009
C06074=1041.007,19.248,-82.972,169.524,37.258,157.009
C06075=1041.001,18.999,-82.955,169.522,37.257,157.009
C06076=1040.995,18.750,-82.940,169.520,37.256,157.008
C06077=1040.988,18.500,-82.925,169.518,37.255,157.008
C06078=1040.982,18.250,-82.908,169.516,37.255,157.008
C06079=1040.975,18.001,-82.893,169.513,37.253,157.008
C06080=1040.969,17.751,-82.877,169.511,37.253,157.008
C06081=1040.963,17.502,-82.861,169.509,37.252,157.008
C06082=1040.956,17.253,-82.846,169.508,37.252,157.008
C06083=1040.950,17.003,-82.830,169.506,37.250,157.007
C06084=1040.944,16.754,-82.814,169.504,37.250,157.007
C06085=1040.938,16.505,-82.798,169.502,37.249,157.007
C06086=1040.931,16.255,-82.783,169.500,37.249,157.007
C06087=1040.925,16.006,-82.768,169.498,37.247,157.007
C06088=1040.919,15.756,-82.752,169.496,37.247,157.007
C06089=1040.912,15.507,-82.736,169.493,37.246,157.006
C06090=1040.906,15.258,-82.721,169.491,37.245,157.006
C06091=1040.900,15.008,-82.705,169.489,37.244,157.006
C06092=1040.893,14.759,-82.690,169.488,37.244,157.006
C06093=1040.888,14.509,-82.674,169.486,37.243,157.006
C06094=1040.881,14.260,-82.658,169.484,37.242,157.006
C06095=1040.874,14.010,-82.643,169.482,37.241,157.005
C06096=1040.868,13.761,-82.628,169.480,37.241,157.005
C06097=1040.862,13.511,-82.612,169.478,37.240,157.005
C06098=1040.855,13.262,-82.596,169.475,37.239,157.005
C06099=1040.845,12.862,-82.572,169.472,37.238,157.005
C06100=1040.834,12.462,-82.548,169.469,37.237,157.005
C06101=1040.824,12.062,-82.523,169.466,37.236,157.004
C06102=1040.814,11.662,-82.498,169.463,37.235,157.004
C06103=1040.807,11.412,-82.483,169.461,37.234,157.004
C06104=1040.801,11.163,-82.468,169.459,37.233,157.004
C06105=1040.794,10.914,-82.453,169.457,37.233,157.004
C06106=1040.788,10.665,-82.437,169.454,37.232,157.004
C06107=1040.782,10.415,-82.421,169.452,37.231,157.003
C06108=1040.776,10.165,-82.406,169.450,37.231,157.003
C06109=1040.769,9.916,-82.391,169.448,37.230,157.003
C06110=1040.763,9.666,-82.376,169.446,37.229,157.003
C06111=1040.756,9.417,-82.360,169.444,37.228,157.003
C06112=1040.750,9.168,-82.345,169.442,37.228,157.003
C06113=1040.743,8.918,-82.330,169.440,37.227,157.003
C06114=1040.736,8.669,-82.315,169.438,37.227,157.002
C06115=1040.730,8.419,-82.300,169.436,37.226,157.002
C06116=1040.724,8.169,-82.284,169.433,37.225,157.002
C06117=1040.718,7.920,-82.269,169.431,37.225,157.002
C06118=1040.711,7.671,-82.254,169.429,37.224,157.002
C06119=1040.705,7.421,-82.239,169.428,37.223,157.002
C06120=1040.699,7.171,-82.224,169.426,37.222,157.002
C06121=1040.692,6.922,-82.208,169.424,37.222,157.001
C06122=1040.685,6.673,-82.193,169.422,37.221,157.001
C06123=1040.680,6.424,-82.178,169.420,37.221,157.001
C06124=1040.673,6.174,-82.164,169.418,37.219,157.001
C06125=1040.667,5.925,-82.148,169.415,37.219,157.001
C06126=1040.660,5.675,-82.133,169.413,37.218,157.001
C06127=1040.655,5.425,-82.117,169.411,37.217,157.001
C06128=1040.648,5.176,-82.102,169.409,37.217,157.000
C06129=1040.642,4.927,-82.087,169.407,37.216,157.000
C06130=1040.635,4.677,-82.072,169.405,37.216,157.000
C06131=1040.629,4.427,-82.057,169.403,37.214,157.000
C06132=1040.623,4.178,-82.042,169.401,37.214,157.000
C06133=1040.617,3.929,-82.027,169.399,37.213,157.000
C06134=1040.610,3.680,-82.012,169.397,37.213,157.000
C06135=1040.604,3.430,-81.997,169.395,37.212,156.999
C06136=1040.597,3.180,-81.982,169.392,37.211,156.999
C06137=1040.591,2.931,-81.967,169.390,37.210,156.999
C06138=1040.584,2.681,-81.952,169.388,37.210,156.999
C06139=1040.579,2.432,-81.937,169.386,37.209,156.999
C06140=1040.572,2.183,-81.922,169.384,37.208,156.999
C06141=1040.566,1.933,-81.907,169.382,37.208,156.999
C06142=1040.560,1.683,-81.891,169.380,37.207,156.998
C06143=1040.554,1.434,-81.876,169.378,37.207,156.998
C06144=1040.548,1.185,-81.862,169.377,37.205,156.998
C06145=1040.541,0.935,-81.847,169.374,37.205,156.998
C06146=1040.535,0.685,-81.832,169.372,37.204,156.998
C06147=1040.529,0.436,-81.817,169.370,37.203,156.998
C06148=1040.522,0.186,-81.802,169.368,37.203,156.998
C06149=1040.516,-0.063,-81.787,169.366,37.202,156.997
C06150=1040.510,-0.312,-81.772,169.364,37.201,156.997
C06151=1040.503,-0.562,-81.757,169.362,37.200,156.997
C06152=1040.497,-0.811,-81.742,169.360,37.200,156.997
C06153=1040.491,-1.061,-81.727,169.358,37.199,156.997
C06154=1040.485,-1.310,-81.712,169.356,37.199,156.997
C06155=1040.475,-1.694,-81.689,169.352,37.197,156.996
C06156=1040.466,-2.079,-81.666,169.349,37.196,156.996
C06157=1040.456,-2.463,-81.644,169.346,37.195,156.996
C06158=1040.447,-2.848,-81.621,169.343,37.194,156.996
C06159=1040.439,-3.131,-81.604,169.340,37.193,156.996
C06160=1040.432,-3.414,-81.587,169.338,37.192,156.995
C06161=1040.425,-3.698,-81.571,169.336,37.192,156.995
C06162=1040.417,-3.981,-81.554,169.333,37.191,156.995
C06163=1040.412,-4.231,-81.540,169.331,37.191,156.995
C06164=1040.405,-4.480,-81.525,169.328,37.190,156.995
C06165=1040.399,-4.730,-81.510,169.326,37.189,156.995
C06166=1040.392,-4.979,-81.495,169.324,37.189,156.995
C06167=1040.386,-5.228,-81.481,169.322,37.188,156.995
C06168=1040.380,-5.478,-81.466,169.320,37.188,156.994
C06169=1040.373,-5.727,-81.452,169.318,37.187,156.994
C06170=1040.367,-5.978,-81.437,169.316,37.186,156.994
C06171=1040.361,-6.227,-81.423,169.314,37.186,156.994
C06172=1040.354,-6.476,-81.408,169.312,37.185,156.994
C06173=1040.347,-6.726,-81.393,169.310,37.185,156.994
C06174=1040.341,-6.975,-81.379,169.308,37.184,156.994
C06175=1040.335,-7.225,-81.365,169.305,37.183,156.994
C06176=1040.328,-7.474,-81.350,169.303,37.183,156.993
C06177=1040.322,-7.724,-81.335,169.301,37.182,156.993
C06178=1040.316,-7.973,-81.321,169.299,37.182,156.993
C06179=1040.309,-8.223,-81.307,169.297,37.181,156.993
C06180=1040.303,-8.472,-81.292,169.295,37.180,156.993
C06181=1040.297,-8.722,-81.277,169.293,37.180,156.993
C06182=1040.291,-8.971,-81.263,169.291,37.179,156.993
C06183=1040.284,-9.221,-81.249,169.289,37.179,156.993
C06184=1040.278,-9.471,-81.234,169.287,37.178,156.992
C06185=1040.272,-9.720,-81.219,169.285,37.177,156.992
C06186=1040.265,-9.970,-81.206,169.282,37.177,156.992
C06187=1040.259,-10.219,-81.191,169.280,37.176,156.992
C06188=1040.253,-10.468,-81.176,169.278,37.176,156.992
C06189=1040.246,-10.718,-81.163,169.275,37.175,156.992
C06190=1040.240,-10.967,-81.148,169.273,37.174,156.992
C06191=1040.234,-11.217,-81.133,169.271,37.174,156.992
C06192=1040.227,-11.467,-81.120,169.269,37.173,156.991
C06193=1040.221,-11.716,-81.105,169.267,37.172,156.991
C06194=1040.215,-11.965,-81.090,169.265,37.172,156.991
C06195=1040.208,-12.215,-81.076,169.263,37.171,156.991
C06196=1040.202,-12.464,-81.062,169.261,37.171,156.991
C06197=1040.196,-12.714,-81.047,169.259,37.170,156.991
C06198=1040.190,-12.963,-81.034,169.256,37.169,156.991
C06199=1040.183,-13.213,-81.019,169.254,37.169,156.990
C06200=1040.177,-13.463,-81.004,169.252,37.168,156.990
C06201=1040.171,-13.712,-80.990,169.250,37.168,156.990
C06202=1040.165,-13.962,-80.976,169.248,37.167,156.990
C06203=1040.159,-14.211,-80.962,169.246,37.166,156.990
C06204=1040.152,-14.460,-80.947,169.244,37.166,156.990
C06205=1040.146,-14.710,-80.933,169.242,37.165,156.990
C06206=1040.139,-14.959,-80.919,169.240,37.165,156.990
C06207=1040.134,-15.209,-80.905,169.237,37.164,156.989
C06208=1040.127,-15.459,-80.890,169.235,37.164,156.989
C06209=1040.120,-15.708,-80.877,169.233,37.163,156.989
C06210=1040.114,-15.957,-80.863,169.230,37.163,156.989
C06211=1040.108,-16.207,-80.848,169.228,37.162,156.989
C06212=1040.102,-16.457,-80.835,169.226,37.162,156.989
C06213=1040.095,-16.706,-80.820,169.224,37.161,156.989
C06214=1040.088,-16.956,-80.807,169.222,37.161,156.989
C06215=1040.083,-17.205,-80.792,169.220,37.160,156.989
C06216=1040.076,-17.455,-80.778,169.218,37.160,156.989
C06217=1040.069,-17.704,-80.764,169.215,37.159,156.988
C06218=1040.063,-17.954,-80.750,169.213,37.159,156.988
C06219=1040.057,-18.203,-80.737,169.211,37.158,156.988
C06220=1040.051,-18.453,-80.722,169.209,37.158,156.988
C06221=1040.044,-18.702,-80.709,169.207,37.157,156.988
C06222=1040.038,-18.952,-80.695,169.205,37.157,156.988
C06223=1040.030,-19.234,-80.679,169.202,37.156,156.988
C06224=1040.023,-19.515,-80.663,169.199,37.156,156.988
C06225=1040.017,-19.798,-80.647,169.197,37.155,156.988
C06226=1040.009,-20.080,-80.631,169.194,37.154,156.987
C06227=1040.003,-20.329,-80.618,169.192,37.154,156.987
C06228=1039.996,-20.578,-80.603,169.190,37.153,156.987
C06229=1039.990,-20.828,-80.590,169.188,37.153,156.987
C06230=1039.984,-21.078,-80.576,169.186,37.153,156.987
C06231=1039.977,-21.327,-80.563,169.184,37.152,156.987
C06232=1039.972,-21.576,-80.548,169.182,37.151,156.987
C06233=1039.965,-21.826,-80.534,169.179,37.151,156.987
C06234=1039.959,-22.076,-80.521,169.177,37.150,156.987
C06235=1039.952,-22.325,-80.506,169.175,37.150,156.987
C06236=1039.946,-22.574,-80.493,169.173,37.150,156.986
C06237=1039.940,-22.825,-80.479,169.170,37.149,156.986
C06238=1039.934,-23.074,-80.465,169.168,37.148,156.986
C06239=1039.927,-23.324,-80.452,169.166,37.148,156.986
C06240=1039.921,-23.573,-80.437,169.164,37.148,156.986
C06241=1039.915,-23.822,-80.424,169.161,37.147,156.986
C06242=1039.909,-24.072,-80.410,169.159,37.147,156.986
C06243=1039.903,-24.322,-80.396,169.157,37.146,156.986
C06244=1039.896,-24.572,-80.383,169.155,37.145,156.986
C06245=1039.890,-24.821,-80.368,169.153,37.145,156.985
C06246=1039.883,-25.070,-80.355,169.151,37.145,156.985
C06247=1039.877,-25.320,-80.341,169.149,37.144,156.985
C06248=1039.871,-25.569,-80.327,169.146,37.144,156.985
C06249=1039.865,-25.819,-80.314,169.144,37.143,156.985
C06250=1039.858,-26.069,-80.301,169.142,37.142,156.985
C06251=1039.853,-26.317,-80.286,169.139,37.142,156.985
C06252=1039.846,-26.567,-80.272,169.137,37.142,156.985
C06253=1039.840,-26.817,-80.259,169.135,37.141,156.985
C06254=1039.833,-27.067,-80.245,169.133,37.141,156.985
C06255=1039.827,-27.316,-80.232,169.130,37.140,156.984
C06256=1039.821,-27.566,-80.218,169.128,37.140,156.984
C06257=1039.814,-27.815,-80.205,169.126,37.139,156.984
C06258=1039.808,-28.065,-80.191,169.124,37.139,156.984
C06259=1039.801,-28.315,-80.178,169.122,37.139,156.984
C06260=1039.795,-28.564,-80.165,169.120,37.138,156.984
C06261=1039.789,-28.813,-80.151,169.117,37.138,156.984
C06262=1039.783,-29.064,-80.137,169.115,37.138,156.984
C06263=1039.777,-29.313,-80.124,169.113,37.137,156.984
C06264=1039.770,-29.562,-80.110,169.111,37.136,156.984
C06265=1039.763,-29.812,-80.097,169.109,37.136,156.984
C06266=1039.757,-30.061,-80.084,169.106,37.136,156.983
C06267=1039.750,-30.311,-80.070,169.103,37.135,156.983
C06268=1039.744,-30.561,-80.057,169.101,37.135,156.983
C06269=1039.738,-30.810,-80.043,169.099,37.135,156.983
C06270=1039.731,-31.060,-80.030,169.097,37.134,156.983
C06271=1039.725,-31.309,-80.016,169.094,37.134,156.983
C06272=1039.719,-31.558,-80.003,169.092,37.133,156.983
C06273=1039.713,-31.808,-79.991,169.090,37.133,156.983
C06274=1039.707,-32.058,-79.976,169.088,37.133,156.983
C06275=1039.701,-32.308,-79.963,169.086,37.132,156.983
C06276=1039.694,-32.557,-79.950,169.083,37.132,156.983
C06277=1039.688,-32.807,-79.936,169.081,37.132,156.983
C06278=1039.681,-33.056,-79.923,169.079,37.131,156.982
C06279=1039.675,-33.305,-79.910,169.077,37.130,156.982
C06280=1039.668,-33.555,-79.896,169.075,37.131,156.982
C06281=1039.662,-33.805,-79.884,169.072,37.130,156.982
C06282=1039.656,-34.055,-79.870,169.070,37.129,156.982
C06283=1039.650,-34.304,-79.857,169.068,37.129,156.982
C06284=1039.643,-34.554,-79.843,169.065,37.129,156.982
C06285=1039.637,-34.803,-79.830,169.063,37.129,156.982
C06286=1039.631,-35.053,-79.818,169.060,37.128,156.982
C06287=1039.624,-35.334,-79.802,169.058,37.128,156.982
C06288=1039.617,-35.615,-79.787,169.055,37.127,156.982
C06289=1039.610,-35.896,-79.772,169.053,37.127,156.982
C06290=1039.603,-36.177,-79.758,169.050,37.126,156.981
C06291=1039.597,-36.427,-79.744,169.048,37.126,156.981
C06292=1039.591,-36.676,-79.731,169.046,37.126,156.981
C06293=1039.584,-36.926,-79.717,169.044,37.125,156.981
C06294=1039.578,-37.176,-79.705,169.042,37.125,156.981
C06295=1039.572,-37.425,-79.692,169.039,37.125,156.981
C06296=1039.565,-37.674,-79.678,169.037,37.124,156.981
C06297=1039.560,-37.924,-79.666,169.035,37.123,156.981
C06298=1039.553,-38.173,-79.652,169.033,37.123,156.981
C06299=1039.547,-38.423,-79.639,169.031,37.123,156.981
C06300=1039.541,-38.673,-79.626,169.028,37.123,156.981
C06301=1039.534,-38.922,-79.613,169.026,37.122,156.981
C06302=1039.528,-39.172,-79.600,169.023,37.122,156.980
C06303=1039.522,-39.422,-79.587,169.021,37.122,156.980
C06304=1039.515,-39.672,-79.574,169.018,37.121,156.980
C06305=1039.509,-39.921,-79.561,169.016,37.121,156.980
C06306=1039.503,-40.170,-79.548,169.014,37.121,156.980
C06307=1039.496,-40.420,-79.535,169.011,37.121,156.980
C06308=1039.490,-40.670,-79.522,169.009,37.121,156.980
C06309=1039.484,-40.920,-79.509,169.007,37.120,156.980
C06310=1039.477,-41.169,-79.497,169.005,37.120,156.980
C06311=1039.471,-41.418,-79.484,169.002,37.119,156.980
C06312=1039.465,-41.668,-79.470,169.000,37.119,156.980
C06313=1039.459,-41.917,-79.458,168.998,37.119,156.980
C06314=1039.452,-42.167,-79.445,168.996,37.119,156.980
C06315=1039.446,-42.416,-79.433,168.993,37.118,156.980
C06316=1039.439,-42.666,-79.419,168.991,37.118,156.980
C06317=1039.433,-42.916,-79.406,168.989,37.118,156.979
C06318=1039.427,-43.165,-79.393,168.987,37.118,156.979
C06319=1039.420,-43.415,-79.381,168.984,37.117,156.979
C06320=1039.414,-43.664,-79.368,168.982,37.117,156.979
C06321=1039.408,-43.914,-79.355,168.980,37.117,156.979
C06322=1039.402,-44.164,-79.343,168.977,37.117,156.979
C06323=1039.395,-44.413,-79.330,168.975,37.116,156.979
C06324=1039.389,-44.663,-79.318,168.973,37.116,156.979
C06325=1039.383,-44.913,-79.304,168.971,37.116,156.979
C06326=1039.377,-45.163,-79.291,168.967,37.115,156.979
C06327=1039.370,-45.412,-79.278,168.965,37.115,156.979
C06328=1039.364,-45.662,-79.266,168.963,37.115,156.979
C06329=1039.358,-45.911,-79.254,168.960,37.115,156.979
C06330=1039.352,-46.161,-79.240,168.958,37.114,156.979
C06331=1039.346,-46.411,-79.228,168.956,37.114,156.979
C06332=1039.339,-46.660,-79.215,168.954,37.114,156.978
C06333=1039.333,-46.909,-79.203,168.951,37.114,156.978
C06334=1039.327,-47.159,-79.190,168.949,37.113,156.978
C06335=1039.320,-47.408,-79.177,168.947,37.113,156.978
C06336=1039.314,-47.658,-79.165,168.944,37.113,156.978
C06337=1039.308,-47.908,-79.152,168.942,37.113,156.978
C06338=1039.302,-48.157,-79.139,168.940,37.113,156.978
C06339=1039.295,-48.407,-79.127,168.938,37.112,156.978
C06340=1039.289,-48.657,-79.114,168.935,37.112,156.978
C06341=1039.283,-48.906,-79.101,168.933,37.111,156.978
C06342=1039.277,-49.156,-79.089,168.931,37.111,156.978
C06343=1039.271,-49.405,-79.077,168.928,37.111,156.978
C06344=1039.264,-49.655,-79.063,168.926,37.111,156.978
C06345=1039.259,-49.905,-79.051,168.924,37.110,156.978
C06346=1039.252,-50.154,-79.039,168.921,37.110,156.978
C06347=1039.246,-50.404,-79.026,168.919,37.110,156.978
C06348=1039.240,-50.653,-79.013,168.917,37.110,156.978
C06349=1039.233,-50.903,-79.001,168.914,37.110,156.978
C06350=1039.227,-51.153,-78.989,168.912,37.110,156.978
C06351=1039.219,-51.435,-78.975,168.909,37.110,156.978
C06352=1039.212,-51.716,-78.961,168.906,37.109,156.977
C06353=1039.206,-51.997,-78.948,168.903,37.109,156.977
C06354=1039.198,-52.279,-78.933,168.900,37.109,156.977
C06355=1039.192,-52.528,-78.921,168.898,37.109,156.977
C06356=1039.185,-52.778,-78.909,168.896,37.109,156.977
C06357=1039.179,-53.028,-78.897,168.893,37.109,156.977
C06358=1039.172,-53.277,-78.885,168.891,37.109,156.977
C06359=1039.167,-53.527,-78.872,168.889,37.109,156.977
C06360=1039.160,-53.777,-78.860,168.886,37.109,156.977
C06361=1039.153,-54.026,-78.848,168.884,37.109,156.977
C06362=1039.147,-54.276,-78.836,168.882,37.108,156.977
C06363=1039.140,-54.525,-78.823,168.879,37.108,156.977
C06364=1039.134,-54.775,-78.811,168.877,37.108,156.977
C06365=1039.128,-55.025,-78.799,168.874,37.108,156.977
C06366=1039.121,-55.274,-78.787,168.872,37.108,156.977
C06367=1039.115,-55.524,-78.775,168.870,37.108,156.977
C06368=1039.109,-55.774,-78.762,168.867,37.108,156.977
C06369=1039.103,-56.023,-78.750,168.865,37.108,156.977
C06370=1039.097,-56.272,-78.738,168.863,37.108,156.977
C06371=1039.090,-56.522,-78.726,168.860,37.108,156.977
C06372=1039.083,-56.772,-78.714,168.858,37.108,156.977
C06373=1039.077,-57.021,-78.701,168.855,37.107,156.977
C06374=1039.071,-57.271,-78.689,168.853,37.107,156.977
C06375=1039.064,-57.521,-78.678,168.851,37.107,156.977
C06376=1039.059,-57.771,-78.666,168.848,37.108,156.977
C06377=1039.052,-58.021,-78.654,168.846,37.108,156.977
C06378=1039.046,-58.270,-78.642,168.843,37.108,156.977
C06379=1039.040,-58.519,-78.630,168.841,37.107,156.977
C06380=1039.033,-58.769,-78.618,168.839,37.107,156.977
C06381=1039.027,-59.019,-78.606,168.836,37.107,156.977
C06382=1039.021,-59.268,-78.593,168.834,37.107,156.977
C06383=1039.014,-59.518,-78.581,168.832,37.107,156.977
C06384=1039.007,-59.768,-78.569,168.829,37.107,156.977
C06385=1039.001,-60.016,-78.558,168.827,37.107,156.976
C06386=1038.996,-60.267,-78.546,168.824,37.107,156.976
C06387=1038.989,-60.517,-78.534,168.822,37.107,156.976
C06388=1038.983,-60.766,-78.522,168.820,37.107,156.976
C06389=1038.977,-61.016,-78.509,168.817,37.107,156.976
C06390=1038.971,-61.265,-78.498,168.815,37.107,156.976
C06391=1038.964,-61.514,-78.486,168.812,37.107,156.976
C06392=1038.958,-61.765,-78.474,168.810,37.107,156.976
C06393=1038.952,-62.014,-78.462,168.808,37.106,156.976
C06394=1038.945,-62.264,-78.450,168.805,37.106,156.976
C06395=1038.940,-62.513,-78.438,168.803,37.106,156.976
C06396=1038.933,-62.763,-78.426,168.800,37.106,156.976
C06397=1038.927,-63.013,-78.415,168.798,37.106,156.976
C06398=1038.920,-63.263,-78.403,168.796,37.106,156.976
C06399=1038.915,-63.512,-78.390,168.793,37.106,156.976
C06400=1038.908,-63.761,-78.378,168.791,37.106,156.976
C06401=1038.902,-64.012,-78.367,168.788,37.106,156.976
C06402=1038.896,-64.261,-78.355,168.786,37.106,156.976
C06403=1038.890,-64.510,-78.343,168.784,37.106,156.976
C06404=1038.883,-64.760,-78.331,168.781,37.106,156.976
C06405=1038.877,-65.010,-78.320,168.778,37.106,156.976
C06406=1038.872,-65.259,-78.308,168.775,37.106,156.976
C06407=1038.865,-65.509,-78.296,168.773,37.106,156.976
C06408=1038.859,-65.759,-78.285,168.771,37.106,156.976
C06409=1038.852,-66.009,-78.273,168.768,37.106,156.976
C06410=1038.847,-66.258,-78.260,168.766,37.106,156.976
C06411=1038.840,-66.508,-78.249,168.763,37.106,156.976
C06412=1038.834,-66.758,-78.237,168.761,37.106,156.976
C06413=1038.828,-67.006,-78.226,168.758,37.106,156.976
C06414=1038.822,-67.257,-78.214,168.756,37.106,156.976
C06415=1038.815,-67.540,-78.201,168.753,37.106,156.976
C06416=1038.808,-67.822,-78.187,168.751,37.106,156.976
C06417=1038.801,-68.105,-78.174,168.748,37.106,156.976
C06418=1038.794,-68.388,-78.161,168.745,37.105,156.976
C06419=1038.788,-68.638,-78.149,168.743,37.105,156.976
C06420=1038.782,-68.887,-78.138,168.740,37.105,156.976
C06421=1038.776,-69.137,-78.125,168.738,37.105,156.976
C06422=1038.769,-69.387,-78.114,168.735,37.105,156.976
C06423=1038.763,-69.636,-78.102,168.733,37.105,156.976
C06424=1038.757,-69.886,-78.091,168.731,37.105,156.976
C06425=1038.752,-70.135,-78.079,168.728,37.106,156.976
C06426=1038.745,-70.385,-78.068,168.726,37.106,156.976
C06427=1038.739,-70.635,-78.056,168.723,37.106,156.976
C06428=1038.733,-70.884,-78.045,168.721,37.106,156.976
C06429=1038.726,-71.134,-78.033,168.718,37.106,156.976
C06430=1038.721,-71.384,-78.021,168.716,37.105,156.975
C06431=1038.715,-71.633,-78.010,168.714,37.105,156.975
C06432=1038.709,-71.883,-77.999,168.711,37.105,156.975
C06433=1038.702,-72.132,-77.987,168.709,37.105,156.975
C06434=1038.697,-72.383,-77.975,168.706,37.105,156.975
C06435=1038.691,-72.632,-77.963,168.704,37.105,156.975
C06436=1038.684,-72.882,-77.952,168.701,37.105,156.975
C06437=1038.679,-73.131,-77.941,168.699,37.105,156.975
C06438=1038.672,-73.381,-77.929,168.696,37.105,156.975
C06439=1038.667,-73.631,-77.918,168.694,37.105,156.975
C06440=1038.660,-73.880,-77.906,168.692,37.105,156.975
C06441=1038.655,-74.130,-77.895,168.689,37.105,156.975
C06442=1038.648,-74.380,-77.884,168.687,37.106,156.975
C06443=1038.642,-74.629,-77.872,168.684,37.106,156.975
C06444=1038.636,-74.879,-77.861,168.682,37.106,156.975
C06445=1038.630,-75.129,-77.850,168.679,37.106,156.975
C06446=1038.623,-75.378,-77.838,168.677,37.106,156.975
C06447=1038.617,-75.628,-77.827,168.674,37.106,156.975
C06448=1038.611,-75.878,-77.816,168.672,37.106,156.975
C06449=1038.605,-76.128,-77.805,168.669,37.106,156.975
C06450=1038.598,-76.377,-77.794,168.667,37.106,156.975
C06451=1038.592,-76.627,-77.782,168.664,37.107,156.975
C06452=1038.586,-76.876,-77.771,168.662,37.107,156.975
C06453=1038.580,-77.126,-77.760,168.659,37.107,156.975
C06454=1038.574,-77.375,-77.749,168.657,37.107,156.975
C06455=1038.567,-77.625,-77.737,168.654,37.107,156.975
C06456=1038.562,-77.875,-77.727,168.652,37.107,156.975
C06457=1038.555,-78.125,-77.715,168.649,37.107,156.975
C06458=1038.549,-78.374,-77.704,168.647,37.107,156.975
C06459=1038.543,-78.624,-77.692,168.644,37.108,156.975
C06460=1038.537,-78.874,-77.682,168.642,37.108,156.975
C06461=1038.532,-79.123,-77.671,168.639,37.108,156.975
C06462=1038.525,-79.373,-77.659,168.637,37.108,156.975
C06463=1038.519,-79.623,-77.649,168.634,37.108,156.975
C06464=1038.512,-79.872,-77.637,168.632,37.108,156.975
C06465=1038.506,-80.122,-77.626,168.629,37.109,156.975
C06466=1038.500,-80.372,-77.615,168.627,37.109,156.975
C06467=1038.494,-80.621,-77.604,168.624,37.109,156.975
C06468=1038.487,-80.871,-77.594,168.622,37.110,156.976
C06469=1038.481,-81.121,-77.583,168.619,37.110,156.976
C06470=1038.475,-81.371,-77.571,168.617,37.111,156.976
C06471=1038.469,-81.620,-77.561,168.614,37.111,156.976
C06472=1038.462,-81.870,-77.550,168.612,37.111,156.976
C06473=1038.457,-82.120,-77.539,168.609,37.111,156.976
C06474=1038.450,-82.369,-77.529,168.606,37.111,156.976
C06475=1038.444,-82.619,-77.517,168.604,37.111,156.976
C06476=1038.438,-82.869,-77.507,168.601,37.112,156.976
C06477=1038.431,-83.118,-77.496,168.599,37.112,156.976
C06478=1038.425,-83.368,-77.485,168.596,37.112,156.976
C06479=1038.418,-83.653,-77.473,168.594,37.113,156.976
C06480=1038.411,-83.937,-77.460,168.591,37.113,156.976
C06481=1038.403,-84.223,-77.448,168.589,37.114,156.976
C06482=1038.396,-84.508,-77.436,168.586,37.114,156.976
C06483=1038.390,-84.758,-77.425,168.583,37.114,156.976
C06484=1038.385,-85.007,-77.414,168.581,37.114,156.976
C06485=1038.378,-85.257,-77.403,168.578,37.114,156.976
C06486=1038.372,-85.506,-77.392,168.575,37.115,156.976
C06487=1038.365,-85.756,-77.382,168.573,37.115,156.976
C06488=1038.359,-86.006,-77.371,168.570,37.115,156.976
C06489=1038.354,-86.256,-77.361,168.568,37.116,156.976
C06490=1038.347,-86.506,-77.350,168.565,37.116,156.976
C06491=1038.341,-86.755,-77.339,168.563,37.117,156.976
C06492=1038.335,-87.005,-77.328,168.560,37.117,156.976
C06493=1038.328,-87.255,-77.318,168.558,37.117,156.976
C06494=1038.322,-87.504,-77.307,168.555,37.117,156.976
C06495=1038.317,-87.754,-77.296,168.552,37.117,156.976
C06496=1038.310,-88.003,-77.286,168.550,37.118,156.977
C06497=1038.304,-88.254,-77.275,168.547,37.118,156.977
C06498=1038.297,-88.503,-77.265,168.545,37.119,156.977
C06499=1038.292,-88.752,-77.254,168.542,37.119,156.977
C06500=1038.285,-89.002,-77.243,168.540,37.119,156.977
C06501=1038.279,-89.252,-77.233,168.537,37.120,156.977
C06502=1038.273,-89.502,-77.222,168.535,37.120,156.977
C06503=1038.267,-89.751,-77.212,168.532,37.120,156.977
C06504=1038.261,-90.001,-77.201,168.529,37.120,156.977
C06505=1038.255,-90.251,-77.190,168.527,37.121,156.977
C06506=1038.249,-90.500,-77.180,168.524,37.121,156.977
C06507=1038.243,-90.750,-77.169,168.522,37.121,156.977
C06508=1038.237,-91.000,-77.158,168.519,37.122,156.977
C06509=1038.231,-91.250,-77.148,168.517,37.122,156.977
C06510=1038.225,-91.499,-77.138,168.514,37.123,156.977
C06511=1038.218,-91.749,-77.127,168.511,37.123,156.977
C06512=1038.212,-91.999,-77.117,168.509,37.123,156.977
C06513=1038.206,-92.249,-77.106,168.506,37.123,156.977
C06514=1038.200,-92.498,-77.096,168.505,37.124,156.977
C06515=1038.194,-92.747,-77.085,168.502,37.124,156.977
C06516=1038.188,-92.997,-77.075,168.500,37.125,156.977
C06517=1038.182,-93.247,-77.064,168.497,37.125,156.977
C06518=1038.176,-93.497,-77.054,168.494,37.126,156.977
C06519=1038.170,-93.747,-77.043,168.492,37.126,156.977
C06520=1038.164,-93.996,-77.033,168.489,37.126,156.977
C06521=1038.158,-94.246,-77.023,168.487,37.126,156.978
C06522=1038.152,-94.496,-77.012,168.484,37.126,156.978
C06523=1038.145,-94.745,-77.001,168.482,37.127,156.978
C06524=1038.140,-94.996,-76.991,168.479,37.127,156.978
C06525=1038.133,-95.245,-76.981,168.476,37.128,156.978
C06526=1038.128,-95.495,-76.971,168.474,37.128,156.978
C06527=1038.121,-95.744,-76.961,168.471,37.129,156.978
C06528=1038.116,-95.993,-76.950,168.469,37.129,156.978
C06529=1038.110,-96.244,-76.940,168.466,37.129,156.978
C06530=1038.104,-96.493,-76.929,168.463,37.129,156.978
C06531=1038.098,-96.744,-76.919,168.461,37.130,156.978
C06532=1038.091,-96.993,-76.908,168.458,37.130,156.978
C06533=1038.086,-97.243,-76.898,168.456,37.131,156.978
C06534=1038.079,-97.492,-76.888,168.453,37.131,156.978
C06535=1038.074,-97.742,-76.878,168.451,37.132,156.978
C06536=1038.067,-97.991,-76.868,168.448,37.132,156.978
C06537=1038.061,-98.241,-76.858,168.445,37.133,156.978
C06538=1038.056,-98.491,-76.848,168.443,37.133,156.978
C06539=1038.049,-98.740,-76.838,168.440,37.134,156.978
C06540=1038.042,-98.991,-76.828,168.437,37.134,156.979
C06541=1038.037,-99.240,-76.817,168.435,37.134,156.979
C06542=1038.031,-99.490,-76.807,168.433,37.135,156.979
C06543=1038.023,-99.778,-76.796,168.430,37.136,156.979
C06544=1038.017,-100.064,-76.784,168.427,37.137,156.979
C06545=1038.010,-100.351,-76.773,168.424,37.137,156.979
C06546=1038.002,-100.638,-76.761,168.421,37.137,156.979
C06547=1037.997,-100.889,-76.751,168.418,37.138,156.979
C06548=1037.990,-101.138,-76.741,168.416,37.139,156.979
C06549=1037.984,-101.388,-76.731,168.413,37.139,156.979
C06550=1037.978,-101.637,-76.722,168.411,37.140,156.979
C06551=1037.972,-101.887,-76.711,168.408,37.140,156.979
C06552=1037.966,-102.137,-76.701,168.405,37.141,156.979
C06553=1037.959,-102.387,-76.691,168.403,37.141,156.979
C06554=1037.954,-102.637,-76.680,168.400,37.142,156.980
C06555=1037.948,-102.886,-76.671,168.397,37.142,156.980
C06556=1037.941,-103.136,-76.661,168.395,37.143,156.980
C06557=1037.935,-103.386,-76.652,168.392,37.143,156.980
///RCONF 1,0,0,0,1,0,0,0,0,0,0,0,0,0,0,0,0,0,0,0,0,0,0,0
C06558=1037.929,-103.636,-76.641,168.390,37.144,156.980
C06559=1037.923,-103.885,-76.631,168.387,37.145,156.980
C06560=1037.917,-104.135,-76.622,168.385,37.145,156.980
C06561=1037.911,-104.385,-76.612,168.383,37.145,156.980
C06562=1037.905,-104.634,-76.601,168.380,37.146,156.980
C06563=1037.899,-104.884,-76.592,168.377,37.147,156.980
C06564=1037.893,-105.134,-76.582,168.375,37.147,156.980
C06565=1037.887,-105.383,-76.573,168.372,37.148,156.980
C06566=1037.882,-105.633,-76.563,168.369,37.148,156.980
C06567=1037.876,-105.883,-76.553,168.367,37.149,156.981
C06568=1037.869,-106.132,-76.543,168.364,37.150,156.981
C06569=1037.863,-106.382,-76.533,168.361,37.150,156.981
C06570=1037.857,-106.632,-76.524,168.359,37.151,156.981
C06571=1037.851,-106.882,-76.514,168.356,37.151,156.981
C06572=1037.845,-107.132,-76.504,168.353,37.152,156.981
C06573=1037.839,-107.381,-76.495,168.351,37.152,156.981
C06574=1037.833,-107.631,-76.485,168.348,37.153,156.981
C06575=1037.827,-107.881,-76.475,168.346,37.154,156.981
C06576=1037.820,-108.130,-76.465,168.343,37.154,156.981
C06577=1037.814,-108.380,-76.456,168.341,37.155,156.981
C06578=1037.808,-108.630,-76.446,168.338,37.156,156.982
C06579=1037.802,-108.880,-76.436,168.336,37.157,156.982
C06580=1037.796,-109.130,-76.426,168.333,37.157,156.982
C06581=1037.790,-109.380,-76.417,168.330,37.158,156.982
C06582=1037.785,-109.629,-76.407,168.328,37.158,156.982
C06583=1037.778,-109.878,-76.398,168.325,37.159,156.982
C06584=1037.772,-110.128,-76.388,168.322,37.159,156.982
C06585=1037.766,-110.378,-76.379,168.320,37.160,156.982
C06586=1037.760,-110.628,-76.369,168.317,37.161,156.982
C06587=1037.754,-110.878,-76.360,168.314,37.162,156.982
C06588=1037.748,-111.127,-76.350,168.312,37.162,156.982
C06589=1037.741,-111.377,-76.341,168.309,37.163,156.983
C06590=1037.736,-111.626,-76.331,168.306,37.164,156.983
C06591=1037.730,-111.876,-76.322,168.304,37.164,156.983
C06592=1037.724,-112.127,-76.313,168.302,37.165,156.983
C06593=1037.718,-112.376,-76.303,168.299,37.166,156.983
C06594=1037.711,-112.626,-76.294,168.297,37.167,156.983
C06595=1037.705,-112.876,-76.284,168.294,37.167,156.983
C06596=1037.699,-113.126,-76.275,168.291,37.168,156.983
C06597=1037.693,-113.375,-76.265,168.289,37.169,156.983
C06598=1037.687,-113.625,-76.256,168.286,37.169,156.983
C06599=1037.681,-113.874,-76.246,168.283,37.170,156.984
C06600=1037.675,-114.124,-76.237,168.281,37.171,156.984
C06601=1037.669,-114.375,-76.228,168.278,37.171,156.984
C06602=1037.664,-114.624,-76.219,168.275,37.172,156.984
C06603=1037.657,-114.874,-76.209,168.273,37.173,156.984
C06604=1037.651,-115.123,-76.200,168.270,37.174,156.984
C06605=1037.645,-115.373,-76.190,168.267,37.174,156.984
C06606=1037.639,-115.623,-76.180,168.265,37.175,156.984
C06607=1037.633,-115.909,-76.170,168.262,37.176,156.984
C06608=1037.625,-116.195,-76.160,168.259,37.177,156.985
C06609=1037.619,-116.482,-76.149,168.256,37.178,156.985
C06610=1037.612,-116.768,-76.138,168.253,37.179,156.985
C06611=1037.605,-117.018,-76.130,168.250,37.179,156.985
C06612=1037.599,-117.268,-76.120,168.248,37.181,156.985
C06613=1037.594,-117.517,-76.111,168.245,37.181,156.985
C06614=1037.587,-117.767,-76.101,168.242,37.182,156.985
C06615=1037.581,-118.018,-76.092,168.240,37.183,156.985
C06616=1037.575,-118.267,-76.083,168.237,37.183,156.985
C06617=1037.570,-118.516,-76.074,168.234,37.184,156.986
C06618=1037.564,-118.767,-76.065,168.232,37.185,156.986
C06619=1037.557,-119.016,-76.056,168.230,37.186,156.986
C06620=1037.551,-119.266,-76.046,168.227,37.187,156.986
C06621=1037.546,-119.516,-76.038,168.224,37.188,156.986
C06622=1037.539,-119.766,-76.028,168.222,37.188,156.986
C06623=1037.533,-120.015,-76.019,168.219,37.189,156.986
C06624=1037.528,-120.265,-76.010,168.216,37.190,156.986
C06625=1037.521,-120.515,-76.001,168.213,37.191,156.987
C06626=1037.515,-120.764,-75.992,168.211,37.192,156.987
C06627=1037.510,-121.014,-75.983,168.208,37.193,156.987
C06628=1037.503,-121.264,-75.974,168.205,37.193,156.987
C06629=1037.498,-121.514,-75.965,168.204,37.194,156.987
C06630=1037.491,-121.763,-75.956,168.201,37.195,156.987
C06631=1037.485,-122.014,-75.947,168.198,37.196,156.987
C06632=1037.479,-122.263,-75.938,168.195,37.197,156.987
C06633=1037.474,-122.512,-75.929,168.193,37.197,156.988
C06634=1037.468,-122.763,-75.920,168.190,37.198,156.988
C06635=1037.461,-123.012,-75.911,168.187,37.200,156.988
C06636=1037.456,-123.262,-75.902,168.184,37.200,156.988
C06637=1037.449,-123.512,-75.893,168.182,37.201,156.988
C06638=1037.444,-123.762,-75.884,168.179,37.202,156.988
C06639=1037.438,-124.011,-75.875,168.176,37.203,156.988
C06640=1037.431,-124.262,-75.866,168.175,37.204,156.988
C06641=1037.426,-124.511,-75.857,168.172,37.204,156.989
C06642=1037.420,-124.761,-75.848,168.169,37.206,156.989
C06643=1037.413,-125.011,-75.839,168.166,37.207,156.989
C06644=1037.408,-125.260,-75.831,168.164,37.207,156.989
C06645=1037.402,-125.511,-75.822,168.161,37.209,156.989
C06646=1037.396,-125.759,-75.813,168.158,37.209,156.989
C06647=1037.390,-126.010,-75.805,168.155,37.210,156.989
C06648=1037.384,-126.260,-75.795,168.153,37.211,156.990
C06649=1037.378,-126.509,-75.787,168.150,37.212,156.990
C06650=1037.372,-126.760,-75.778,168.148,37.213,156.990
C06651=1037.366,-127.009,-75.769,168.145,37.214,156.990
C06652=1037.360,-127.259,-75.761,168.143,37.215,156.990
C06653=1037.354,-127.508,-75.752,168.140,37.216,156.990
C06654=1037.347,-127.758,-75.743,168.137,37.217,156.990
C06655=1037.342,-128.007,-75.734,168.135,37.218,156.990
C06656=1037.338,-128.257,-75.724,168.132,37.218,156.990
C06657=1037.333,-128.507,-75.715,168.130,37.218,156.990
C06658=1037.330,-128.757,-75.704,168.127,37.217,156.990
C06659=1037.327,-129.007,-75.692,168.125,37.216,156.990
C06660=1037.326,-129.256,-75.680,168.124,37.215,156.990
C06661=1037.325,-129.507,-75.667,168.121,37.212,156.989
C06662=1037.324,-129.756,-75.654,168.119,37.210,156.989
C06663=1037.325,-130.007,-75.640,168.118,37.207,156.988
C06664=1037.326,-130.256,-75.626,168.116,37.203,156.988
C06665=1037.327,-130.507,-75.611,168.115,37.200,156.987
C06666=1037.331,-130.757,-75.596,168.113,37.196,156.987
C06667=1037.334,-131.007,-75.579,168.112,37.190,156.986
C06668=1037.339,-131.257,-75.563,168.110,37.185,156.985
C06669=1037.343,-131.508,-75.545,168.109,37.180,156.984
C06670=1037.350,-131.757,-75.527,168.109,37.174,156.983
C06671=1037.010,-131.781,-75.799,168.061,37.382,157.017
C06672=1037.005,-131.532,-75.816,168.061,37.388,157.018
C06673=1037.000,-131.282,-75.834,168.062,37.394,157.019
C06674=1036.995,-131.032,-75.851,168.064,37.399,157.020
C06675=1036.992,-130.781,-75.867,168.065,37.404,157.021
C06676=1036.989,-130.531,-75.882,168.067,37.408,157.022
C06677=1036.988,-130.281,-75.898,168.068,37.411,157.022
C06678=1036.986,-130.031,-75.912,168.070,37.415,157.023
C06679=1036.985,-129.781,-75.925,168.071,37.418,157.024
C06680=1036.985,-129.531,-75.939,168.074,37.421,157.024
C06681=1036.986,-129.281,-75.952,168.075,37.423,157.024
C06682=1036.988,-129.032,-75.963,168.077,37.424,157.025
C06683=1036.991,-128.781,-75.975,168.079,37.425,157.025
C06684=1036.994,-128.531,-75.986,168.082,37.426,157.025
C06685=1036.998,-128.281,-75.996,168.084,37.426,157.025
C06686=1037.003,-128.032,-76.006,168.086,37.426,157.025
C06687=1037.008,-127.783,-76.016,168.089,37.425,157.025
C06688=1037.014,-127.533,-76.024,168.092,37.424,157.025
C06689=1037.020,-127.283,-76.032,168.095,37.423,157.025
C06690=1037.026,-127.034,-76.041,168.097,37.422,157.025
C06691=1037.032,-126.784,-76.050,168.100,37.421,157.024
C06692=1037.038,-126.533,-76.059,168.103,37.420,157.024
C06693=1037.044,-126.284,-76.067,168.106,37.419,157.024
C06694=1037.050,-126.034,-76.076,168.107,37.419,157.024
C06695=1037.056,-125.785,-76.085,168.110,37.417,157.024
C06696=1037.062,-125.535,-76.094,168.113,37.416,157.024
C06697=1037.068,-125.284,-76.102,168.116,37.415,157.024
C06698=1037.074,-125.035,-76.112,168.118,37.414,157.023
C06699=1037.080,-124.785,-76.120,168.121,37.414,157.023
C06700=1037.086,-124.536,-76.129,168.124,37.412,157.023
C06701=1037.092,-124.286,-76.138,168.127,37.411,157.023
C06702=1037.099,-124.036,-76.147,168.129,37.411,157.023
C06703=1037.104,-123.786,-76.155,168.131,37.409,157.023
C06704=1037.110,-123.537,-76.165,168.134,37.409,157.023
C06705=1037.115,-123.287,-76.174,168.137,37.408,157.023
C06706=1037.122,-123.037,-76.183,168.139,37.406,157.022
C06707=1037.128,-122.787,-76.191,168.142,37.406,157.022
C06708=1037.134,-122.538,-76.201,168.145,37.405,157.022
C06709=1037.140,-122.288,-76.209,168.148,37.404,157.022
C06710=1037.146,-122.038,-76.219,168.150,37.403,157.022
C06711=1037.152,-121.788,-76.227,168.153,37.402,157.022
C06712=1037.158,-121.539,-76.236,168.156,37.401,157.022
C06713=1037.164,-121.288,-76.245,168.159,37.401,157.022
C06714=1037.169,-121.039,-76.254,168.160,37.399,157.021
C06715=1037.176,-120.789,-76.264,168.163,37.399,157.021
C06716=1037.182,-120.539,-76.272,168.166,37.398,157.021
C06717=1037.188,-120.290,-76.281,168.168,37.397,157.021
C06718=1037.194,-120.040,-76.291,168.171,37.396,157.021
C06719=1037.200,-119.790,-76.300,168.174,37.395,157.021
C06720=1037.205,-119.541,-76.309,168.177,37.394,157.021
C06721=1037.211,-119.290,-76.318,168.179,37.394,157.021
C06722=1037.218,-119.041,-76.327,168.182,37.393,157.020
C06723=1037.224,-118.791,-76.336,168.185,37.391,157.020
C06724=1037.230,-118.541,-76.345,168.187,37.391,157.020
C06725=1037.236,-118.292,-76.355,168.189,37.390,157.020
C06726=1037.242,-118.042,-76.364,168.192,37.389,157.020
C06727=1037.247,-117.792,-76.373,168.195,37.389,157.020
C06728=1037.253,-117.542,-76.382,168.198,37.387,157.020
C06729=1037.260,-117.293,-76.391,168.200,37.386,157.020
C06730=1037.266,-117.043,-76.401,168.203,37.386,157.019
C06731=1037.272,-116.793,-76.409,168.206,37.385,157.019
C06732=1037.278,-116.507,-76.420,168.209,37.384,157.019
C06733=1037.285,-116.220,-76.431,168.212,37.383,157.019
C06734=1037.293,-115.934,-76.441,168.215,37.382,157.019
C06735=1037.299,-115.647,-76.452,168.218,37.381,157.019
C06736=1037.305,-115.397,-76.462,168.220,37.381,157.019
C06737=1037.312,-115.147,-76.471,168.223,37.380,157.019
C06738=1037.317,-114.898,-76.480,168.225,37.379,157.018
C06739=1037.323,-114.649,-76.490,168.228,37.378,157.018
C06740=1037.330,-114.398,-76.498,168.231,37.377,157.018
C06741=1037.336,-114.149,-76.508,168.233,37.376,157.018
C06742=1037.342,-113.899,-76.517,168.236,37.376,157.018
C06743=1037.348,-113.650,-76.527,168.239,37.375,157.018
C06744=1037.353,-113.400,-76.537,168.242,37.374,157.018
C06745=1037.360,-113.150,-76.546,168.244,37.374,157.018
C06746=1037.366,-112.900,-76.556,168.247,37.373,157.018
C06747=1037.372,-112.650,-76.565,168.250,37.372,157.018
C06748=1037.377,-112.401,-76.574,168.251,37.371,157.017
C06749=1037.383,-112.151,-76.583,168.254,37.371,157.017
C06750=1037.389,-111.901,-76.593,168.257,37.370,157.017
C06751=1037.396,-111.651,-76.603,168.259,37.369,157.017
C06752=1037.402,-111.401,-76.612,168.262,37.368,157.017
C06753=1037.408,-111.152,-76.622,168.265,37.368,157.017
C06754=1037.414,-110.902,-76.631,168.268,37.367,157.017
C06755=1037.420,-110.653,-76.641,168.270,37.366,157.017
C06756=1037.426,-110.403,-76.650,168.273,37.366,157.017
C06757=1037.432,-110.153,-76.660,168.276,37.365,157.017
C06758=1037.438,-109.903,-76.669,168.278,37.364,157.017
C06759=1037.444,-109.654,-76.679,168.281,37.363,157.016
C06760=1037.451,-109.404,-76.688,168.284,37.363,157.016
C06761=1037.457,-109.154,-76.698,168.285,37.362,157.016
C06762=1037.463,-108.904,-76.707,168.288,37.361,157.016
C06763=1037.469,-108.654,-76.717,168.291,37.361,157.016
C06764=1037.475,-108.405,-76.726,168.293,37.360,157.016
C06765=1037.480,-108.155,-76.736,168.296,37.359,157.016
C06766=1037.486,-107.905,-76.746,168.299,37.358,157.016
C06767=1037.492,-107.656,-76.756,168.302,37.358,157.016
C06768=1037.499,-107.406,-76.765,168.304,37.357,157.016
C06769=1037.505,-107.156,-76.775,168.307,37.356,157.015
C06770=1037.511,-106.907,-76.785,168.310,37.356,157.015
C06771=1037.517,-106.657,-76.795,168.312,37.355,157.015
C06772=1037.523,-106.407,-76.805,168.315,37.355,157.015
C06773=1037.529,-106.157,-76.814,168.318,37.354,157.015
C06774=1037.535,-105.907,-76.824,168.320,37.353,157.015
C06775=1037.541,-105.657,-76.833,168.323,37.353,157.015
C06776=1037.548,-105.408,-76.843,168.325,37.352,157.015
C06777=1037.553,-105.158,-76.854,168.327,37.351,157.015
C06778=1037.559,-104.908,-76.863,168.330,37.350,157.015
C06779=1037.566,-104.659,-76.873,168.333,37.350,157.015
C06780=1037.572,-104.409,-76.883,168.335,37.350,157.015
C06781=1037.577,-104.159,-76.893,168.338,37.349,157.014
C06782=1037.584,-103.909,-76.903,168.340,37.348,157.014
C06783=1037.590,-103.660,-76.913,168.343,37.348,157.014
C06784=1037.596,-103.410,-76.922,168.346,37.347,157.014
C06785=1037.601,-103.160,-76.932,168.348,37.347,157.014
C06786=1037.608,-102.911,-76.943,168.351,37.346,157.014
C06787=1037.614,-102.661,-76.952,168.354,37.345,157.014
C06788=1037.620,-102.411,-76.962,168.356,37.345,157.014
C06789=1037.626,-102.161,-76.972,168.359,37.345,157.014
C06790=1037.632,-101.912,-76.982,168.362,37.344,157.014
C06791=1037.638,-101.662,-76.992,168.364,37.343,157.014
///RCONF 1,0,0,0,0,0,0,0,0,0,0,0,0,0,0,0,0,0,0,0,0,0,0,0
C06792=1037.644,-101.412,-77.002,168.367,37.342,157.014
C06793=1037.650,-101.163,-77.012,168.370,37.342,157.014
C06794=1037.656,-100.913,-77.022,168.371,37.342,157.014
C06795=1037.663,-100.663,-77.031,168.374,37.341,157.013
C06796=1037.670,-100.376,-77.044,168.377,37.340,157.013
C06797=1037.677,-100.089,-77.055,168.380,37.339,157.013
C06798=1037.684,-99.801,-77.066,168.383,37.339,157.013
C06799=1037.690,-99.514,-77.078,168.386,37.338,157.013
C06800=1037.697,-99.265,-77.088,168.389,37.338,157.013
C06801=1037.703,-99.015,-77.098,168.391,37.337,157.013
C06802=1037.709,-98.765,-77.108,168.394,37.336,157.013
C06803=1037.715,-98.515,-77.118,168.397,37.336,157.013
C06804=1037.721,-98.266,-77.128,168.399,37.336,157.013
C06805=1037.727,-98.016,-77.139,168.402,37.335,157.013
C06806=1037.733,-97.766,-77.148,168.405,37.334,157.013
C06807=1037.740,-97.517,-77.159,168.407,37.334,157.013
C06808=1037.745,-97.267,-77.169,168.410,37.334,157.013
C06809=1037.752,-97.018,-77.179,168.412,37.333,157.012
C06810=1037.758,-96.767,-77.190,168.415,37.333,157.012
C06811=1037.764,-96.518,-77.200,168.418,37.332,157.012
C06812=1037.770,-96.268,-77.210,168.420,37.332,157.012
C06813=1037.775,-96.018,-77.221,168.422,37.331,157.012
C06814=1037.782,-95.769,-77.231,168.424,37.331,157.012
C06815=1037.787,-95.519,-77.241,168.427,37.330,157.012
C06816=1037.794,-95.269,-77.251,168.430,37.330,157.012
C06817=1037.799,-95.020,-77.262,168.432,37.330,157.012
C06818=1037.806,-94.770,-77.273,168.435,37.329,157.012
C06819=1037.812,-94.520,-77.283,168.437,37.329,157.012
C06820=1037.817,-94.270,-77.294,168.440,37.328,157.012
C06821=1037.824,-94.020,-77.303,168.443,37.328,157.012
C06822=1037.829,-93.771,-77.314,168.445,37.327,157.012
C06823=1037.836,-93.522,-77.324,168.448,37.327,157.012
C06824=1037.841,-93.272,-77.334,168.450,37.327,157.012
C06825=1037.848,-93.022,-77.345,168.453,37.327,157.012
C06826=1037.854,-92.772,-77.356,168.456,37.326,157.012
C06827=1037.860,-92.522,-77.366,168.458,37.326,157.012
C06828=1037.866,-92.273,-77.376,168.461,37.325,157.012
C06829=1037.872,-92.024,-77.387,168.463,37.325,157.012
C06830=1037.879,-91.773,-77.397,168.466,37.324,157.011
C06831=1037.884,-91.524,-77.408,168.469,37.324,157.011
C06832=1037.890,-91.274,-77.419,168.471,37.324,157.011
C06833=1037.896,-91.024,-77.429,168.474,37.324,157.011
C06834=1037.903,-90.774,-77.440,168.476,37.323,157.011
C06835=1037.909,-90.525,-77.450,168.479,37.323,157.011
C06836=1037.915,-90.275,-77.461,168.481,37.322,157.011
C06837=1037.920,-90.025,-77.471,168.484,37.322,157.011
C06838=1037.927,-89.776,-77.481,168.487,37.321,157.011
C06839=1037.933,-89.526,-77.493,168.489,37.321,157.011
C06840=1037.940,-89.277,-77.503,168.492,37.321,157.011
C06841=1037.945,-89.027,-77.513,168.494,37.321,157.011
C06842=1037.951,-88.776,-77.524,168.496,37.320,157.011
C06843=1037.958,-88.527,-77.535,168.499,37.320,157.011
C06844=1037.963,-88.278,-77.546,168.501,37.319,157.011
C06845=1037.970,-88.029,-77.556,168.504,37.319,157.011
C06846=1037.976,-87.778,-77.566,168.506,37.318,157.011
C06847=1037.982,-87.528,-77.577,168.509,37.318,157.011
C06848=1037.988,-87.279,-77.588,168.511,37.318,157.011
C06849=1037.995,-87.029,-77.599,168.514,37.317,157.011
C06850=1038.000,-86.779,-77.610,168.517,37.317,157.011
C06851=1038.007,-86.530,-77.620,168.519,37.317,157.011
C06852=1038.013,-86.280,-77.631,168.522,37.317,157.011
C06853=1038.019,-86.030,-77.641,168.524,37.316,157.011
C06854=1038.025,-85.781,-77.652,168.527,37.316,157.011
C06855=1038.031,-85.531,-77.663,168.529,37.315,157.010
C06856=1038.038,-85.281,-77.673,168.532,37.315,157.010
C06857=1038.044,-85.032,-77.684,168.535,37.314,157.010
C06858=1038.050,-84.782,-77.695,168.537,37.314,157.010
C06859=1038.056,-84.533,-77.706,168.540,37.314,157.010
C06860=1038.064,-84.247,-77.718,168.543,37.314,157.010
C06861=1038.070,-83.963,-77.730,168.546,37.313,157.010
C06862=1038.077,-83.677,-77.743,168.548,37.313,157.010
C06863=1038.085,-83.392,-77.756,168.551,37.313,157.010
C06864=1038.091,-83.143,-77.766,168.554,37.312,157.010
C06865=1038.097,-82.894,-77.777,168.557,37.312,157.010
C06866=1038.103,-82.643,-77.788,168.559,37.311,157.010
C06867=1038.110,-82.394,-77.798,168.562,37.311,157.010
C06868=1038.116,-82.144,-77.810,168.564,37.310,157.010
C06869=1038.122,-81.894,-77.820,168.567,37.310,157.010
C06870=1038.129,-81.645,-77.831,168.569,37.310,157.010
C06871=1038.135,-81.395,-77.842,168.572,37.310,157.010
C06872=1038.140,-81.146,-77.853,168.574,37.310,157.010
C06873=1038.147,-80.896,-77.864,168.577,37.309,157.010
C06874=1038.153,-80.646,-77.874,168.580,37.309,157.010
C06875=1038.160,-80.396,-77.886,168.582,37.309,157.010
C06876=1038.166,-80.147,-77.896,168.584,37.308,157.010
C06877=1038.172,-79.897,-77.907,168.586,37.308,157.010
C06878=1038.178,-79.647,-77.918,168.589,37.308,157.010
C06879=1038.184,-79.397,-77.929,168.591,37.307,157.010
C06880=1038.190,-79.147,-77.940,168.594,37.307,157.010
C06881=1038.197,-78.898,-77.952,168.596,37.307,157.010
C06882=1038.203,-78.648,-77.963,168.599,37.307,157.010
C06883=1038.209,-78.398,-77.974,168.601,37.307,157.010
C06884=1038.215,-78.149,-77.985,168.604,37.306,157.010
C06885=1038.222,-77.899,-77.996,168.606,37.306,157.010
C06886=1038.228,-77.650,-78.007,168.609,37.306,157.010
C06887=1038.233,-77.401,-78.018,168.611,37.306,157.010
C06888=1038.240,-77.150,-78.029,168.614,37.305,157.010
C06889=1038.246,-76.901,-78.040,168.616,37.305,157.010
C06890=1038.252,-76.651,-78.052,168.619,37.305,157.010
C06891=1038.258,-76.402,-78.063,168.621,37.305,157.010
C06892=1038.264,-76.152,-78.074,168.624,37.305,157.010
C06893=1038.271,-75.901,-78.086,168.626,37.305,157.009
C06894=1038.277,-75.653,-78.097,168.629,37.305,157.009
C06895=1038.283,-75.402,-78.109,168.631,37.304,157.009
C06896=1038.289,-75.153,-78.119,168.634,37.304,157.010
C06897=1038.295,-74.903,-78.131,168.636,37.304,157.010
C06898=1038.301,-74.654,-78.142,168.639,37.304,157.009
C06899=1038.307,-74.404,-78.153,168.641,37.304,157.009
C06900=1038.314,-74.155,-78.164,168.644,37.304,157.009
C06901=1038.320,-73.905,-78.176,168.646,37.304,157.009
C06902=1038.326,-73.655,-78.187,168.649,37.303,157.009
C06903=1038.332,-73.405,-78.199,168.651,37.303,157.009
C06904=1038.338,-73.156,-78.210,168.654,37.303,157.010
C06905=1038.344,-72.906,-78.221,168.656,37.303,157.010
C06906=1038.350,-72.656,-78.234,168.659,37.303,157.010
C06907=1038.356,-72.406,-78.245,168.661,37.303,157.010
C06908=1038.363,-72.157,-78.257,168.664,37.303,157.010
C06909=1038.368,-71.907,-78.268,168.666,37.303,157.010
C06910=1038.375,-71.658,-78.280,168.668,37.303,157.010
C06911=1038.380,-71.408,-78.291,168.671,37.303,157.010
C06912=1038.387,-71.158,-78.303,168.673,37.303,157.010
C06913=1038.392,-70.909,-78.314,168.676,37.303,157.010
C06914=1038.399,-70.659,-78.326,168.678,37.303,157.010
C06915=1038.405,-70.409,-78.338,168.681,37.303,157.010
C06916=1038.411,-70.160,-78.349,168.683,37.303,157.010
C06917=1038.417,-69.910,-78.360,168.686,37.303,157.010
C06918=1038.423,-69.661,-78.372,168.688,37.303,157.010
C06919=1038.429,-69.410,-78.384,168.690,37.303,157.010
C06920=1038.435,-69.161,-78.396,168.693,37.303,157.010
C06921=1038.441,-68.911,-78.407,168.695,37.302,157.010
C06922=1038.448,-68.662,-78.419,168.698,37.302,157.010
C06923=1038.454,-68.413,-78.430,168.700,37.302,157.010
C06924=1038.460,-68.129,-78.444,168.703,37.302,157.010
C06925=1038.467,-67.847,-78.457,168.706,37.302,157.010
C06926=1038.474,-67.564,-78.470,168.708,37.302,157.010
C06927=1038.481,-67.280,-78.484,168.711,37.302,157.010
C06928=1038.487,-67.032,-78.495,168.715,37.303,157.010
C06929=1038.494,-66.781,-78.506,168.717,37.303,157.010
C06930=1038.500,-66.532,-78.518,168.720,37.303,157.010
C06931=1038.506,-66.283,-78.531,168.722,37.303,157.010
C06932=1038.512,-66.032,-78.542,168.724,37.303,157.010
C06933=1038.519,-65.783,-78.554,168.727,37.302,157.010
C06934=1038.525,-65.534,-78.565,168.729,37.302,157.010
C06935=1038.530,-65.284,-78.577,168.732,37.302,157.010
C06936=1038.537,-65.034,-78.589,168.734,37.302,157.010
C06937=1038.543,-64.785,-78.601,168.737,37.302,157.010
C06938=1038.549,-64.535,-78.613,168.739,37.302,157.010
C06939=1038.555,-64.285,-78.625,168.741,37.302,157.010
C06940=1038.562,-64.035,-78.637,168.744,37.302,157.010
C06941=1038.568,-63.787,-78.648,168.746,37.302,157.010
C06942=1038.573,-63.536,-78.660,168.749,37.302,157.010
C06943=1038.580,-63.286,-78.672,168.751,37.302,157.010
C06944=1038.587,-63.037,-78.684,168.753,37.302,157.010
C06945=1038.592,-62.788,-78.696,168.756,37.303,157.010
C06946=1038.598,-62.538,-78.707,168.758,37.302,157.010
C06947=1038.605,-62.288,-78.719,168.761,37.302,157.010
C06948=1038.612,-62.038,-78.731,168.763,37.302,157.010
C06949=1038.617,-61.789,-78.743,168.766,37.302,157.010
C06950=1038.624,-61.540,-78.755,168.768,37.302,157.010
C06951=1038.630,-61.289,-78.767,168.770,37.302,157.010
C06952=1038.636,-61.040,-78.779,168.773,37.302,157.010
C06953=1038.642,-60.790,-78.791,168.775,37.302,157.010
C06954=1038.649,-60.541,-78.803,168.778,37.302,157.010
C06955=1038.654,-60.291,-78.815,168.780,37.302,157.010
C06956=1038.661,-60.042,-78.827,168.782,37.302,157.010
C06957=1038.667,-59.791,-78.838,168.785,37.303,157.011
C06958=1038.674,-59.542,-78.850,168.787,37.303,157.011
C06959=1038.680,-59.292,-78.863,168.790,37.302,157.011
C06960=1038.686,-59.043,-78.875,168.792,37.302,157.011
C06961=1038.693,-58.794,-78.887,168.794,37.302,157.011
C06962=1038.699,-58.544,-78.899,168.797,37.302,157.011
C06963=1038.705,-58.294,-78.911,168.799,37.302,157.011
C06964=1038.712,-58.045,-78.923,168.802,37.302,157.011
C06965=1038.718,-57.795,-78.936,168.804,37.302,157.011
C06966=1038.724,-57.545,-78.948,168.806,37.302,157.011
C06967=1038.730,-57.296,-78.959,168.809,37.303,157.011
C06968=1038.736,-57.046,-78.972,168.811,37.303,157.011
C06969=1038.743,-56.796,-78.983,168.814,37.303,157.011
C06970=1038.749,-56.547,-78.995,168.816,37.303,157.011
C06971=1038.755,-56.297,-79.007,168.818,37.303,157.011
C06972=1038.762,-56.047,-79.019,168.821,37.302,157.011
C06973=1038.769,-55.798,-79.031,168.823,37.302,157.011
C06974=1038.774,-55.548,-79.044,168.826,37.302,157.011
C06975=1038.781,-55.298,-79.056,168.828,37.302,157.011
C06976=1038.787,-55.048,-79.068,168.830,37.303,157.011
C06977=1038.794,-54.799,-79.080,168.833,37.303,157.011
C06978=1038.800,-54.550,-79.093,168.835,37.303,157.011
C06979=1038.806,-54.301,-79.105,168.838,37.303,157.011
C06980=1038.813,-54.051,-79.117,168.840,37.303,157.011
C06981=1038.819,-53.801,-79.129,168.842,37.303,157.011
C06982=1038.825,-53.551,-79.142,168.845,37.303,157.011
C06983=1038.832,-53.302,-79.154,168.847,37.303,157.011
C06984=1038.838,-53.052,-79.166,168.850,37.303,157.011
C06985=1038.844,-52.802,-79.178,168.852,37.303,157.011
C06986=1038.851,-52.553,-79.190,168.854,37.303,157.011
C06987=1038.857,-52.303,-79.203,168.857,37.303,157.011
C06988=1038.865,-52.022,-79.217,168.859,37.303,157.011
C06989=1038.872,-51.740,-79.230,168.862,37.303,157.011
C06990=1038.879,-51.458,-79.245,168.865,37.304,157.011
C06991=1038.886,-51.177,-79.258,168.867,37.303,157.011
C06992=1038.892,-50.928,-79.270,168.870,37.303,157.011
C06993=1038.899,-50.678,-79.282,168.872,37.303,157.011
C06994=1038.905,-50.429,-79.295,168.874,37.303,157.011
C06995=1038.911,-50.179,-79.308,168.878,37.304,157.012
C06996=1038.918,-49.929,-79.320,168.880,37.304,157.012
C06997=1038.924,-49.679,-79.332,168.882,37.304,157.012
C06998=1038.930,-49.430,-79.346,168.885,37.304,157.012
C06999=1038.936,-49.180,-79.358,168.887,37.304,157.012
C07000=1038.943,-48.931,-79.370,168.889,37.304,157.012
C07001=1038.949,-48.681,-79.383,168.892,37.305,157.012
C07002=1038.955,-48.431,-79.396,168.894,37.305,157.012
C07003=1038.961,-48.182,-79.408,168.896,37.305,157.012
C07004=1038.968,-47.933,-79.421,168.899,37.305,157.012
C07005=1038.973,-47.683,-79.434,168.901,37.305,157.012
C07006=1038.979,-47.433,-79.446,168.903,37.306,157.012
C07007=1038.986,-47.184,-79.459,168.906,37.306,157.012
C07008=1038.992,-46.934,-79.471,168.908,37.307,157.012
C07009=1038.998,-46.684,-79.484,168.910,37.306,157.012
C07010=1039.004,-46.435,-79.497,168.912,37.306,157.012
C07011=1039.011,-46.185,-79.509,168.915,37.307,157.012
C07012=1039.018,-45.935,-79.522,168.917,37.307,157.012
C07013=1039.024,-45.685,-79.535,168.919,37.308,157.013
C07014=1039.030,-45.436,-79.548,168.922,37.308,157.013
C07015=1039.037,-45.187,-79.561,168.924,37.307,157.013
C07016=1039.042,-44.937,-79.573,168.926,37.308,157.013
C07017=1039.048,-44.687,-79.586,168.929,37.308,157.013
C07018=1039.055,-44.438,-79.599,168.931,37.309,157.013
C07019=1039.061,-44.188,-79.611,168.933,37.309,157.013
C07020=1039.067,-43.939,-79.624,168.936,37.309,157.013
C07021=1039.073,-43.689,-79.637,168.939,37.309,157.013
C07022=1039.080,-43.440,-79.650,168.941,37.309,157.013
C07023=1039.086,-43.190,-79.663,168.943,37.310,157.013
C07024=1039.093,-42.940,-79.676,168.946,37.310,157.013
C07025=1039.099,-42.690,-79.688,168.948,37.310,157.013
C07026=1039.105,-42.441,-79.701,168.950,37.310,157.013
C07027=1039.111,-42.191,-79.714,168.952,37.310,157.013
C07028=1039.118,-41.942,-79.727,168.955,37.311,157.013
C07029=1039.124,-41.692,-79.739,168.957,37.311,157.013
C07030=1039.130,-41.443,-79.753,168.959,37.311,157.014
C07031=1039.137,-41.192,-79.765,168.962,37.311,157.014
C07032=1039.143,-40.943,-79.779,168.964,37.311,157.014
C07033=1039.150,-40.694,-79.791,168.966,37.312,157.014
C07034=1039.156,-40.444,-79.804,168.968,37.312,157.014
C07035=1039.162,-40.195,-79.817,168.971,37.312,157.014
C07036=1039.168,-39.945,-79.830,168.973,37.312,157.014
C07037=1039.175,-39.695,-79.843,168.975,37.312,157.014
C07038=1039.181,-39.446,-79.855,168.978,37.313,157.014
C07039=1039.188,-39.196,-79.869,168.980,37.313,157.014
C07040=1039.194,-38.947,-79.882,168.982,37.313,157.014
C07041=1039.200,-38.697,-79.894,168.984,37.313,157.014
C07042=1039.206,-38.447,-79.908,168.987,37.314,157.014
C07043=1039.213,-38.198,-79.921,168.989,37.314,157.014
C07044=1039.219,-37.948,-79.934,168.992,37.315,157.014
C07045=1039.225,-37.699,-79.947,168.994,37.314,157.014
C07046=1039.231,-37.450,-79.960,168.997,37.315,157.015
C07047=1039.237,-37.200,-79.973,168.999,37.316,157.015
C07048=1039.244,-36.950,-79.987,169.001,37.316,157.015
C07049=1039.250,-36.700,-80.000,169.003,37.316,157.015
C07050=1039.256,-36.451,-80.013,169.006,37.316,157.015
C07051=1039.262,-36.201,-80.026,169.008,37.317,157.015
C07052=1039.269,-35.920,-80.041,169.010,37.317,157.015
C07053=1039.276,-35.639,-80.056,169.013,37.317,157.015
C07054=1039.283,-35.359,-80.071,169.015,37.318,157.015
C07055=1039.290,-35.077,-80.086,169.018,37.318,157.015
C07056=1039.296,-34.828,-80.099,169.020,37.318,157.015
C07057=1039.303,-34.578,-80.113,169.022,37.319,157.016
C07058=1039.309,-34.328,-80.126,169.024,37.319,157.016
C07059=1039.315,-34.079,-80.138,169.027,37.320,157.016
C07060=1039.321,-33.829,-80.152,169.029,37.320,157.016
C07061=1039.328,-33.579,-80.165,169.032,37.320,157.016
C07062=1039.334,-33.330,-80.179,169.034,37.321,157.016
C07063=1039.341,-33.081,-80.192,169.037,37.321,157.016
C07064=1039.347,-32.831,-80.206,169.039,37.321,157.016
C07065=1039.354,-32.582,-80.219,169.041,37.321,157.016
C07066=1039.360,-32.332,-80.231,169.043,37.322,157.016
C07067=1039.366,-32.082,-80.245,169.045,37.322,157.016
C07068=1039.372,-31.832,-80.259,169.048,37.322,157.016
C07069=1039.378,-31.583,-80.272,169.050,37.323,157.017
C07070=1039.384,-31.334,-80.285,169.052,37.323,157.017
C07071=1039.391,-31.084,-80.299,169.054,37.324,157.017
C07072=1039.397,-30.834,-80.312,169.056,37.324,157.017
C07073=1039.404,-30.585,-80.326,169.059,37.324,157.017
C07074=1039.410,-30.335,-80.339,169.061,37.325,157.017
C07075=1039.417,-30.086,-80.352,169.063,37.325,157.017
C07076=1039.423,-29.837,-80.366,169.065,37.325,157.017
C07077=1039.430,-29.587,-80.379,169.067,37.326,157.017
C07078=1039.436,-29.337,-80.393,169.070,37.326,157.017
C07079=1039.442,-29.088,-80.406,169.073,37.326,157.017
C07080=1039.448,-28.838,-80.420,169.075,37.326,157.017
C07081=1039.454,-28.589,-80.433,169.077,37.327,157.017
C07082=1039.461,-28.339,-80.447,169.079,37.328,157.018
C07083=1039.467,-28.089,-80.460,169.082,37.328,157.018
C07084=1039.474,-27.840,-80.474,169.084,37.328,157.018
C07085=1039.480,-27.590,-80.487,169.086,37.328,157.018
C07086=1039.487,-27.341,-80.500,169.088,37.329,157.018
C07087=1039.493,-27.092,-80.514,169.090,37.329,157.018
C07088=1039.499,-26.841,-80.528,169.093,37.329,157.018
C07089=1039.505,-26.592,-80.541,169.095,37.330,157.018
C07090=1039.512,-26.342,-80.555,169.097,37.330,157.018
C07091=1039.517,-26.093,-80.569,169.099,37.331,157.018
C07092=1039.524,-25.843,-80.582,169.101,37.331,157.018
C07093=1039.530,-25.593,-80.596,169.103,37.332,157.019
C07094=1039.536,-25.344,-80.610,169.107,37.332,157.019
C07095=1039.543,-25.094,-80.624,169.109,37.333,157.019
C07096=1039.549,-24.845,-80.637,169.111,37.333,157.019
C07097=1039.555,-24.596,-80.651,169.113,37.333,157.019
C07098=1039.562,-24.346,-80.665,169.115,37.334,157.019
C07099=1039.568,-24.096,-80.678,169.117,37.335,157.019
C07100=1039.574,-23.847,-80.693,169.119,37.334,157.019
C07101=1039.580,-23.597,-80.706,169.122,37.335,157.019
C07102=1039.587,-23.348,-80.719,169.124,37.336,157.019
C07103=1039.593,-23.098,-80.734,169.126,37.336,157.020
C07104=1039.599,-22.849,-80.748,169.128,37.336,157.020
C07105=1039.605,-22.599,-80.762,169.130,37.337,157.020
C07106=1039.611,-22.350,-80.775,169.132,37.337,157.020
C07107=1039.618,-22.100,-80.789,169.134,37.338,157.020
C07108=1039.624,-21.851,-80.803,169.138,37.339,157.020
C07109=1039.631,-21.601,-80.817,169.140,37.339,157.020
C07110=1039.637,-21.352,-80.830,169.142,37.339,157.020
C07111=1039.643,-21.101,-80.844,169.144,37.340,157.020
C07112=1039.650,-20.853,-80.858,169.146,37.340,157.021
C07113=1039.656,-20.602,-80.873,169.148,37.340,157.021
C07114=1039.662,-20.353,-80.886,169.150,37.341,157.021
C07115=1039.669,-20.104,-80.900,169.153,37.342,157.021
C07116=1039.676,-19.822,-80.915,169.155,37.342,157.021
C07117=1039.683,-19.540,-80.931,169.157,37.343,157.021
C07118=1039.690,-19.257,-80.947,169.160,37.343,157.021
C07119=1039.697,-18.976,-80.963,169.162,37.343,157.021
C07120=1039.703,-18.726,-80.977,169.164,37.344,157.021
C07121=1039.710,-18.478,-80.991,169.166,37.344,157.021
C07122=1039.716,-18.227,-81.005,169.170,37.345,157.022
C07123=1039.723,-17.979,-81.019,169.172,37.345,157.022
C07124=1039.729,-17.728,-81.033,169.174,37.346,157.022
C07125=1039.735,-17.479,-81.047,169.176,37.346,157.022
C07126=1039.742,-17.230,-81.061,169.178,37.347,157.022
C07127=1039.748,-16.980,-81.075,169.180,37.347,157.022
C07128=1039.755,-16.731,-81.089,169.182,37.347,157.022
C07129=1039.761,-16.481,-81.103,169.184,37.348,157.022
C07130=1039.767,-16.231,-81.117,169.187,37.349,157.022
C07131=1039.774,-15.982,-81.131,169.189,37.348,157.022
C07132=1039.779,-15.732,-81.145,169.191,37.349,157.023
C07133=1039.787,-15.483,-81.159,169.193,37.350,157.023
C07134=1039.793,-15.233,-81.173,169.195,37.350,157.023
C07135=1039.799,-14.984,-81.187,169.198,37.351,157.023
C07136=1039.805,-14.734,-81.202,169.200,37.351,157.023
C07137=1039.811,-14.485,-81.216,169.202,37.352,157.023
C07138=1039.818,-14.235,-81.230,169.204,37.352,157.023
C07139=1039.824,-13.986,-81.244,169.206,37.353,157.023
C07140=1039.830,-13.736,-81.259,169.208,37.353,157.023
C07141=1039.837,-13.486,-81.273,169.211,37.354,157.024
C07142=1039.843,-13.237,-81.288,169.213,37.354,157.024
C07143=1039.849,-12.987,-81.302,169.215,37.355,157.024
C07144=1039.855,-12.739,-81.316,169.217,37.356,157.024
C07145=1039.862,-12.489,-81.331,169.219,37.356,157.024
C07146=1039.868,-12.239,-81.345,169.221,37.357,157.024
C07147=1039.874,-11.990,-81.359,169.224,37.357,157.024
C07148=1039.880,-11.740,-81.373,169.226,37.358,157.024
C07149=1039.886,-11.491,-81.388,169.228,37.358,157.024
C07150=1039.893,-11.241,-81.402,169.230,37.359,157.025
C07151=1039.899,-10.991,-81.416,169.232,37.359,157.025
C07152=1039.905,-10.742,-81.431,169.234,37.360,157.025
C07153=1039.912,-10.493,-81.445,169.236,37.360,157.025
C07154=1039.918,-10.243,-81.459,169.238,37.361,157.025
C07155=1039.924,-9.994,-81.474,169.241,37.362,157.025
C07156=1039.931,-9.744,-81.488,169.243,37.362,157.025
C07157=1039.937,-9.494,-81.503,169.245,37.363,157.026
C07158=1039.943,-9.245,-81.517,169.247,37.363,157.026
C07159=1039.950,-8.996,-81.532,169.250,37.364,157.026
C07160=1039.957,-8.746,-81.547,169.252,37.365,157.026
C07161=1039.962,-8.496,-81.560,169.254,37.364,157.026
C07162=1039.969,-8.247,-81.575,169.256,37.365,157.026
C07163=1039.976,-7.997,-81.590,169.258,37.366,157.026
C07164=1039.981,-7.748,-81.604,169.260,37.366,157.026
C07165=1039.988,-7.499,-81.618,169.262,37.367,157.026
C07166=1039.995,-7.249,-81.633,169.264,37.367,157.027
C07167=1040.000,-7.000,-81.647,169.266,37.368,157.027
C07168=1040.007,-6.750,-81.662,169.268,37.369,157.027
C07169=1040.013,-6.500,-81.676,169.270,37.369,157.027
C07170=1040.020,-6.251,-81.691,169.272,37.370,157.027
C07171=1040.026,-6.002,-81.706,169.274,37.370,157.027
C07172=1040.033,-5.752,-81.720,169.277,37.370,157.027
C07173=1040.039,-5.503,-81.735,169.280,37.371,157.027
C07174=1040.046,-5.253,-81.750,169.282,37.372,157.027
C07175=1040.052,-5.004,-81.763,169.284,37.372,157.028
C07176=1040.058,-4.754,-81.778,169.286,37.373,157.028
C07177=1040.065,-4.504,-81.793,169.288,37.373,157.028
C07178=1040.071,-4.255,-81.808,169.290,37.374,157.028
C07179=1040.077,-4.006,-81.822,169.292,37.375,157.028
C07180=1040.085,-3.722,-81.839,169.294,37.375,157.028
C07181=1040.092,-3.438,-81.855,169.296,37.376,157.028
C07182=1040.099,-3.155,-81.873,169.299,37.376,157.028
C07183=1040.106,-2.872,-81.889,169.302,37.377,157.029
C07184=1040.112,-2.622,-81.904,169.304,37.378,157.029
C07185=1040.119,-2.373,-81.919,169.306,37.379,157.029
C07186=1040.124,-2.124,-81.933,169.308,37.379,157.029
C07187=1040.131,-1.874,-81.948,169.310,37.380,157.029
C07188=1040.137,-1.624,-81.963,169.312,37.381,157.029
C07189=1040.144,-1.375,-81.978,169.314,37.381,157.030
C07190=1040.149,-1.126,-81.993,169.316,37.382,157.030
C07191=1040.156,-0.876,-82.008,169.318,37.382,157.030
C07192=1040.162,-0.626,-82.023,169.321,37.383,157.030
C07193=1040.169,-0.377,-82.038,169.323,37.384,157.030
C07194=1040.174,-0.128,-82.052,169.325,37.384,157.030
C07195=1040.180,0.122,-82.068,169.327,37.385,157.030
C07196=1040.186,0.372,-82.083,169.329,37.386,157.031
C07197=1040.193,0.622,-82.098,169.331,37.387,157.031
C07198=1040.199,0.871,-82.113,169.333,37.387,157.031
C07199=1040.205,1.120,-82.128,169.335,37.388,157.031
C07200=1040.212,1.369,-82.143,169.337,37.388,157.031
C07201=1040.218,1.619,-82.158,169.339,37.389,157.031
C07202=1040.224,1.869,-82.173,169.342,37.390,157.031
C07203=1040.231,2.118,-82.188,169.344,37.390,157.031
C07204=1040.237,2.368,-82.203,169.346,37.391,157.032
C07205=1040.243,2.617,-82.217,169.348,37.391,157.032
C07206=1040.249,2.866,-82.232,169.350,37.393,157.032
C07207=1040.256,3.115,-82.248,169.352,37.393,157.032
C07208=1040.262,3.365,-82.263,169.354,37.394,157.032
C07209=1040.269,3.615,-82.278,169.356,37.394,157.032
C07210=1040.275,3.864,-82.293,169.357,37.395,157.032
C07211=1040.281,4.113,-82.307,169.359,37.396,157.033
C07212=1040.288,4.362,-82.323,169.362,37.396,157.033
C07213=1040.293,4.612,-82.338,169.364,37.397,157.033
C07214=1040.300,4.862,-82.353,169.366,37.397,157.033
C07215=1040.306,5.112,-82.368,169.368,37.398,157.033
C07216=1040.312,5.361,-82.383,169.370,37.399,157.033
C07217=1040.319,5.610,-82.399,169.372,37.399,157.033
C07218=1040.325,5.860,-82.414,169.374,37.400,157.034
C07219=1040.332,6.110,-82.429,169.376,37.401,157.034
C07220=1040.338,6.359,-82.443,169.378,37.402,157.034
C07221=1040.344,6.608,-82.459,169.380,37.402,157.034
C07222=1040.351,6.857,-82.474,169.383,37.403,157.034
C07223=1040.357,7.107,-82.489,169.385,37.403,157.034
C07224=1040.363,7.357,-82.504,169.387,37.404,157.034
C07225=1040.369,7.606,-82.520,169.389,37.405,157.035
C07226=1040.376,7.856,-82.535,169.391,37.405,157.035
C07227=1040.382,8.105,-82.550,169.393,37.406,157.035
C07228=1040.389,8.354,-82.566,169.395,37.406,157.035
C07229=1040.395,8.604,-82.581,169.397,37.407,157.035
C07230=1040.402,8.854,-82.596,169.399,37.407,157.035
C07231=1040.408,9.103,-82.611,169.401,37.409,157.035
C07232=1040.415,9.352,-82.626,169.404,37.409,157.036
C07233=1040.421,9.602,-82.641,169.406,37.410,157.036
